(* Logix 5000 project; controller QW361 vendor 1 type 14 code 107 rev 32.11; software revision 32.00; part 11 of 20 *)

        [1429].time.Year := 2022, [1429].time.Month := 4, [1429].time.Day := 28, [1429].time.Hour := 20, [1429].time.Minute := 39, [1429].time.Second := 59, [1429].time.DST_ON := 1, [1430].log_data[0].min := 1.0, [1430].log_data[0].max := 1.0, [1430].log_data[0].total := 300.0, [1430].log_data[0].time := 300.0, [1430].log_data[0].minminute := 40, [1430].log_data[0].maxminute := 40, [1430].log_data[0].valid := 1, [1430].log_data[1].valid := 1, [1430].log_data[2].valid := 1, [1430].log_data[3].valid := 1, [1430].log_data[4].valid := 1, [1430].time.Year := 2022, [1430].time.Month := 4, [1430].time.Day := 28, [1430].time.Hour := 20, [1430].time.Minute := 44, [1430].time.Second := 59, [1430].time.DST_ON := 1, [1431].log_data[0].min := 1.0, [1431].log_data[0].max := 1.0, [1431].log_data[0].total := 300.0, [1431].log_data[0].time := 300.0, [1431].log_data[0].minminute := 45, [1431].log_data[0].maxminute := 45, [1431].log_data[0].valid := 1, [1431].log_data[1].valid := 1, [1431].log_data[2].valid := 1, [1431].log_data[3].valid := 1, [1431].log_data[4].valid := 1, [1431].time.Year := 2022, [1431].time.Month := 4, [1431].time.Day := 28, [1431].time.Hour := 20, [1431].time.Minute := 49, [1431].time.Second := 59, [1431].time.DST_ON := 1, [1432].log_data[0].min := 1.0, [1432].log_data[0].max := 1.0, [1432].log_data[0].total := 300.0, [1432].log_data[0].time := 300.0, [1432].log_data[0].minminute := 50, [1432].log_data[0].maxminute := 50, [1432].log_data[0].valid := 1, [1432].log_data[1].valid := 1, [1432].log_data[2].valid := 1, [1432].log_data[3].valid := 1, [1432].log_data[4].valid := 1, [1432].time.Year := 2022, [1432].time.Month := 4, [1432].time.Day := 28, [1432].time.Hour := 20, [1432].time.Minute := 54, [1432].time.Second := 59,
        [1432].time.DST_ON := 1, [1433].log_data[0].min := 1.0, [1433].log_data[0].max := 1.0, [1433].log_data[0].total := 300.0, [1433].log_data[0].time := 300.0, [1433].log_data[0].minminute := 55, [1433].log_data[0].maxminute := 55, [1433].log_data[0].valid := 1, [1433].log_data[1].valid := 1, [1433].log_data[2].valid := 1, [1433].log_data[3].valid := 1, [1433].log_data[4].valid := 1, [1433].time.Year := 2022, [1433].time.Month := 4, [1433].time.Day := 28, [1433].time.Hour := 20, [1433].time.Minute := 59, [1433].time.Second := 59, [1433].time.DST_ON := 1, [1434].log_data[0].min := 1.0, [1434].log_data[0].max := 1.0, [1434].log_data[0].total := 300.0, [1434].log_data[0].time := 300.0, [1434].log_data[0].valid := 1, [1434].log_data[1].valid := 1, [1434].log_data[2].valid := 1, [1434].log_data[3].valid := 1, [1434].log_data[4].valid := 1, [1434].time.Year := 2022, [1434].time.Month := 4, [1434].time.Day := 28, [1434].time.Hour := 21, [1434].time.Minute := 4, [1434].time.Second := 59, [1434].time.DST_ON := 1, [1435].log_data[0].min := 1.0, [1435].log_data[0].max := 1.0, [1435].log_data[0].total := 300.0, [1435].log_data[0].time := 300.0, [1435].log_data[0].minminute := 5, [1435].log_data[0].maxminute := 5, [1435].log_data[0].valid := 1, [1435].log_data[1].valid := 1, [1435].log_data[2].valid := 1, [1435].log_data[3].valid := 1, [1435].log_data[4].valid := 1, [1435].time.Year := 2022, [1435].time.Month := 4, [1435].time.Day := 28, [1435].time.Hour := 21, [1435].time.Minute := 9, [1435].time.Second := 59, [1435].time.DST_ON := 1, [1436].log_data[0].min := 1.0, [1436].log_data[0].max := 1.0, [1436].log_data[0].total := 300.0, [1436].log_data[0].time := 300.0, [1436].log_data[0].minminute := 10, [1436].log_data[0].maxminute := 10, [1436].log_data[0].valid := 1,
        [1436].log_data[1].valid := 1, [1436].log_data[2].valid := 1, [1436].log_data[3].valid := 1, [1436].log_data[4].valid := 1, [1436].time.Year := 2022, [1436].time.Month := 4, [1436].time.Day := 28, [1436].time.Hour := 21, [1436].time.Minute := 14, [1436].time.Second := 59, [1436].time.DST_ON := 1, [1437].log_data[0].min := 1.0, [1437].log_data[0].max := 1.0, [1437].log_data[0].total := 300.0, [1437].log_data[0].time := 300.0, [1437].log_data[0].minminute := 15, [1437].log_data[0].maxminute := 15, [1437].log_data[0].valid := 1, [1437].log_data[1].valid := 1, [1437].log_data[2].valid := 1, [1437].log_data[3].valid := 1, [1437].log_data[4].valid := 1, [1437].time.Year := 2022, [1437].time.Month := 4, [1437].time.Day := 28, [1437].time.Hour := 21, [1437].time.Minute := 19, [1437].time.Second := 59, [1437].time.DST_ON := 1, [1438].log_data[0].min := 1.0, [1438].log_data[0].max := 1.0, [1438].log_data[0].total := 300.0, [1438].log_data[0].time := 300.0, [1438].log_data[0].minminute := 20, [1438].log_data[0].maxminute := 20, [1438].log_data[0].valid := 1, [1438].log_data[1].valid := 1, [1438].log_data[2].valid := 1, [1438].log_data[3].valid := 1, [1438].log_data[4].valid := 1, [1438].time.Year := 2022, [1438].time.Month := 4, [1438].time.Day := 28, [1438].time.Hour := 21, [1438].time.Minute := 24, [1438].time.Second := 59, [1438].time.DST_ON := 1, [1439].log_data[0].min := 1.0, [1439].log_data[0].max := 1.0, [1439].log_data[0].total := 300.0, [1439].log_data[0].time := 300.0, [1439].log_data[0].minminute := 25, [1439].log_data[0].maxminute := 25, [1439].log_data[0].valid := 1, [1439].log_data[1].valid := 1, [1439].log_data[2].valid := 1, [1439].log_data[3].valid := 1, [1439].log_data[4].valid := 1, [1439].time.Year := 2022, [1439].time.Month := 4,
        [1439].time.Day := 28, [1439].time.Hour := 21, [1439].time.Minute := 29, [1439].time.Second := 59, [1439].time.DST_ON := 1, [1440].log_data[0].min := 1.0, [1440].log_data[0].max := 1.0, [1440].log_data[0].total := 300.0, [1440].log_data[0].time := 300.0, [1440].log_data[0].minminute := 30, [1440].log_data[0].maxminute := 30, [1440].log_data[0].valid := 1, [1440].log_data[1].valid := 1, [1440].log_data[2].valid := 1, [1440].log_data[3].valid := 1, [1440].log_data[4].valid := 1, [1440].time.Year := 2022, [1440].time.Month := 4, [1440].time.Day := 28, [1440].time.Hour := 21, [1440].time.Minute := 34, [1440].time.Second := 59, [1440].time.DST_ON := 1, [1441].log_data[0].min := 1.0, [1441].log_data[0].max := 1.0, [1441].log_data[0].total := 300.0, [1441].log_data[0].time := 300.0, [1441].log_data[0].minminute := 35, [1441].log_data[0].maxminute := 35, [1441].log_data[0].valid := 1, [1441].log_data[1].valid := 1, [1441].log_data[2].valid := 1, [1441].log_data[3].valid := 1, [1441].log_data[4].valid := 1, [1441].time.Year := 2022, [1441].time.Month := 4, [1441].time.Day := 28, [1441].time.Hour := 21, [1441].time.Minute := 39, [1441].time.Second := 59, [1441].time.DST_ON := 1, [1442].log_data[0].min := 1.0, [1442].log_data[0].max := 1.0, [1442].log_data[0].total := 300.0, [1442].log_data[0].time := 300.0, [1442].log_data[0].minminute := 40, [1442].log_data[0].maxminute := 40, [1442].log_data[0].valid := 1, [1442].log_data[1].valid := 1, [1442].log_data[2].valid := 1, [1442].log_data[3].valid := 1, [1442].log_data[4].valid := 1, [1442].time.Year := 2022, [1442].time.Month := 4, [1442].time.Day := 28, [1442].time.Hour := 21, [1442].time.Minute := 44, [1442].time.Second := 59, [1442].time.DST_ON := 1, [1443].log_data[0].min := 1.0,
        [1443].log_data[0].max := 1.0, [1443].log_data[0].total := 300.0, [1443].log_data[0].time := 300.0, [1443].log_data[0].minminute := 45, [1443].log_data[0].maxminute := 45, [1443].log_data[0].valid := 1, [1443].log_data[1].valid := 1, [1443].log_data[2].valid := 1, [1443].log_data[3].valid := 1, [1443].log_data[4].valid := 1, [1443].time.Year := 2022, [1443].time.Month := 4, [1443].time.Day := 28, [1443].time.Hour := 21, [1443].time.Minute := 49, [1443].time.Second := 59, [1443].time.DST_ON := 1, [1444].log_data[0].min := 1.0, [1444].log_data[0].max := 1.0, [1444].log_data[0].total := 300.0, [1444].log_data[0].time := 300.0, [1444].log_data[0].minminute := 50, [1444].log_data[0].maxminute := 50, [1444].log_data[0].valid := 1, [1444].log_data[1].valid := 1, [1444].log_data[2].valid := 1, [1444].log_data[3].valid := 1, [1444].log_data[4].valid := 1, [1444].time.Year := 2022, [1444].time.Month := 4, [1444].time.Day := 28, [1444].time.Hour := 21, [1444].time.Minute := 54, [1444].time.Second := 59, [1444].time.DST_ON := 1, [1445].log_data[0].min := 1.0, [1445].log_data[0].max := 1.0, [1445].log_data[0].total := 300.0, [1445].log_data[0].time := 300.0, [1445].log_data[0].minminute := 55, [1445].log_data[0].maxminute := 55, [1445].log_data[0].valid := 1, [1445].log_data[1].valid := 1, [1445].log_data[2].valid := 1, [1445].log_data[3].valid := 1, [1445].log_data[4].valid := 1, [1445].time.Year := 2022, [1445].time.Month := 4, [1445].time.Day := 28, [1445].time.Hour := 21, [1445].time.Minute := 59, [1445].time.Second := 59, [1445].time.DST_ON := 1, [1446].log_data[0].min := 1.0, [1446].log_data[0].max := 1.0, [1446].log_data[0].total := 300.0, [1446].log_data[0].time := 300.0, [1446].log_data[0].valid := 1, [1446].log_data[1].valid := 1, [1446].log_data[2].valid := 1,
        [1446].log_data[3].valid := 1, [1446].log_data[4].valid := 1, [1446].time.Year := 2022, [1446].time.Month := 4, [1446].time.Day := 28, [1446].time.Hour := 22, [1446].time.Minute := 4, [1446].time.Second := 59, [1446].time.DST_ON := 1, [1447].log_data[0].min := 1.0, [1447].log_data[0].max := 1.0, [1447].log_data[0].total := 300.0, [1447].log_data[0].time := 300.0, [1447].log_data[0].minminute := 5, [1447].log_data[0].maxminute := 5, [1447].log_data[0].valid := 1, [1447].log_data[1].valid := 1, [1447].log_data[2].valid := 1, [1447].log_data[3].valid := 1, [1447].log_data[4].valid := 1, [1447].time.Year := 2022, [1447].time.Month := 4, [1447].time.Day := 28, [1447].time.Hour := 22, [1447].time.Minute := 9, [1447].time.Second := 59, [1447].time.DST_ON := 1, [1448].log_data[0].min := 1.0, [1448].log_data[0].max := 1.0, [1448].log_data[0].total := 300.0, [1448].log_data[0].time := 300.0, [1448].log_data[0].minminute := 10, [1448].log_data[0].maxminute := 10, [1448].log_data[0].valid := 1, [1448].log_data[1].valid := 1, [1448].log_data[2].valid := 1, [1448].log_data[3].valid := 1, [1448].log_data[4].valid := 1, [1448].time.Year := 2022, [1448].time.Month := 4, [1448].time.Day := 28, [1448].time.Hour := 22, [1448].time.Minute := 14, [1448].time.Second := 59, [1448].time.DST_ON := 1, [1449].log_data[0].min := 1.0, [1449].log_data[0].max := 1.0, [1449].log_data[0].total := 300.0, [1449].log_data[0].time := 300.0, [1449].log_data[0].minminute := 15, [1449].log_data[0].maxminute := 15, [1449].log_data[0].valid := 1, [1449].log_data[1].valid := 1, [1449].log_data[2].valid := 1, [1449].log_data[3].valid := 1, [1449].log_data[4].valid := 1, [1449].time.Year := 2022, [1449].time.Month := 4, [1449].time.Day := 28, [1449].time.Hour := 22,
        [1449].time.Minute := 19, [1449].time.Second := 59, [1449].time.DST_ON := 1, [1450].log_data[0].min := 1.0, [1450].log_data[0].max := 1.0, [1450].log_data[0].total := 300.0, [1450].log_data[0].time := 300.0, [1450].log_data[0].minminute := 20, [1450].log_data[0].maxminute := 20, [1450].log_data[0].valid := 1, [1450].log_data[1].valid := 1, [1450].log_data[2].valid := 1, [1450].log_data[3].valid := 1, [1450].log_data[4].valid := 1, [1450].time.Year := 2022, [1450].time.Month := 4, [1450].time.Day := 28, [1450].time.Hour := 22, [1450].time.Minute := 24, [1450].time.Second := 59, [1450].time.DST_ON := 1, [1451].log_data[0].min := 1.0, [1451].log_data[0].max := 1.0, [1451].log_data[0].total := 300.0, [1451].log_data[0].time := 300.0, [1451].log_data[0].minminute := 25, [1451].log_data[0].maxminute := 25, [1451].log_data[0].valid := 1, [1451].log_data[1].valid := 1, [1451].log_data[2].valid := 1, [1451].log_data[3].valid := 1, [1451].log_data[4].valid := 1, [1451].time.Year := 2022, [1451].time.Month := 4, [1451].time.Day := 28, [1451].time.Hour := 22, [1451].time.Minute := 29, [1451].time.Second := 59, [1451].time.DST_ON := 1, [1452].log_data[0].min := 1.0, [1452].log_data[0].max := 1.0, [1452].log_data[0].total := 300.0, [1452].log_data[0].time := 300.0, [1452].log_data[0].minminute := 30, [1452].log_data[0].maxminute := 30, [1452].log_data[0].valid := 1, [1452].log_data[1].valid := 1, [1452].log_data[2].valid := 1, [1452].log_data[3].valid := 1, [1452].log_data[4].valid := 1, [1452].time.Year := 2022, [1452].time.Month := 4, [1452].time.Day := 28, [1452].time.Hour := 22, [1452].time.Minute := 34, [1452].time.Second := 59, [1452].time.DST_ON := 1, [1453].log_data[0].min := 1.0, [1453].log_data[0].max := 1.0, [1453].log_data[0].total := 300.0,
        [1453].log_data[0].time := 300.0, [1453].log_data[0].minminute := 35, [1453].log_data[0].maxminute := 35, [1453].log_data[0].valid := 1, [1453].log_data[1].valid := 1, [1453].log_data[2].valid := 1, [1453].log_data[3].valid := 1, [1453].log_data[4].valid := 1, [1453].time.Year := 2022, [1453].time.Month := 4, [1453].time.Day := 28, [1453].time.Hour := 22, [1453].time.Minute := 39, [1453].time.Second := 59, [1453].time.DST_ON := 1, [1454].log_data[0].min := 1.0, [1454].log_data[0].max := 1.0, [1454].log_data[0].total := 300.0, [1454].log_data[0].time := 300.0, [1454].log_data[0].minminute := 40, [1454].log_data[0].maxminute := 40, [1454].log_data[0].valid := 1, [1454].log_data[1].valid := 1, [1454].log_data[2].valid := 1, [1454].log_data[3].valid := 1, [1454].log_data[4].valid := 1, [1454].time.Year := 2022, [1454].time.Month := 4, [1454].time.Day := 28, [1454].time.Hour := 22, [1454].time.Minute := 44, [1454].time.Second := 59, [1454].time.DST_ON := 1, [1455].log_data[0].min := 1.0, [1455].log_data[0].max := 1.0, [1455].log_data[0].total := 300.0, [1455].log_data[0].time := 300.0, [1455].log_data[0].minminute := 45, [1455].log_data[0].maxminute := 45, [1455].log_data[0].valid := 1, [1455].log_data[1].valid := 1, [1455].log_data[2].valid := 1, [1455].log_data[3].valid := 1, [1455].log_data[4].valid := 1, [1455].time.Year := 2022, [1455].time.Month := 4, [1455].time.Day := 28, [1455].time.Hour := 22, [1455].time.Minute := 49, [1455].time.Second := 59, [1455].time.DST_ON := 1, [1456].log_data[0].min := 1.0, [1456].log_data[0].max := 1.0, [1456].log_data[0].total := 300.0, [1456].log_data[0].time := 300.0, [1456].log_data[0].minminute := 50, [1456].log_data[0].maxminute := 50, [1456].log_data[0].valid := 1, [1456].log_data[1].valid := 1, [1456].log_data[2].valid := 1,
        [1456].log_data[3].valid := 1, [1456].log_data[4].valid := 1, [1456].time.Year := 2022, [1456].time.Month := 4, [1456].time.Day := 28, [1456].time.Hour := 22, [1456].time.Minute := 54, [1456].time.Second := 59, [1456].time.DST_ON := 1, [1457].log_data[0].min := 1.0, [1457].log_data[0].max := 1.0, [1457].log_data[0].total := 300.0, [1457].log_data[0].time := 300.0, [1457].log_data[0].minminute := 55, [1457].log_data[0].maxminute := 55, [1457].log_data[0].valid := 1, [1457].log_data[1].valid := 1, [1457].log_data[2].valid := 1, [1457].log_data[3].valid := 1, [1457].log_data[4].valid := 1, [1457].time.Year := 2022, [1457].time.Month := 4, [1457].time.Day := 28, [1457].time.Hour := 22, [1457].time.Minute := 59, [1457].time.Second := 59, [1457].time.DST_ON := 1, [1458].log_data[0].min := 1.0, [1458].log_data[0].max := 1.0, [1458].log_data[0].total := 300.0, [1458].log_data[0].time := 300.0, [1458].log_data[0].valid := 1, [1458].log_data[1].valid := 1, [1458].log_data[2].valid := 1, [1458].log_data[3].valid := 1, [1458].log_data[4].valid := 1, [1458].time.Year := 2022, [1458].time.Month := 4, [1458].time.Day := 28, [1458].time.Hour := 23, [1458].time.Minute := 4, [1458].time.Second := 59, [1458].time.DST_ON := 1, [1459].log_data[0].min := 1.0, [1459].log_data[0].max := 1.0, [1459].log_data[0].total := 300.0, [1459].log_data[0].time := 300.0, [1459].log_data[0].minminute := 5, [1459].log_data[0].maxminute := 5, [1459].log_data[0].valid := 1, [1459].log_data[1].valid := 1, [1459].log_data[2].valid := 1, [1459].log_data[3].valid := 1, [1459].log_data[4].valid := 1, [1459].time.Year := 2022, [1459].time.Month := 4, [1459].time.Day := 28, [1459].time.Hour := 23, [1459].time.Minute := 9, [1459].time.Second := 59,
        [1459].time.DST_ON := 1, [1460].log_data[0].min := 1.0, [1460].log_data[0].max := 1.0, [1460].log_data[0].total := 300.0, [1460].log_data[0].time := 300.0, [1460].log_data[0].minminute := 10, [1460].log_data[0].maxminute := 10, [1460].log_data[0].valid := 1, [1460].log_data[1].valid := 1, [1460].log_data[2].valid := 1, [1460].log_data[3].valid := 1, [1460].log_data[4].valid := 1, [1460].time.Year := 2022, [1460].time.Month := 4, [1460].time.Day := 28, [1460].time.Hour := 23, [1460].time.Minute := 14, [1460].time.Second := 59, [1460].time.DST_ON := 1, [1461].log_data[0].min := 1.0, [1461].log_data[0].max := 1.0, [1461].log_data[0].total := 300.0, [1461].log_data[0].time := 300.0, [1461].log_data[0].minminute := 15, [1461].log_data[0].maxminute := 15, [1461].log_data[0].valid := 1, [1461].log_data[1].valid := 1, [1461].log_data[2].valid := 1, [1461].log_data[3].valid := 1, [1461].log_data[4].valid := 1, [1461].time.Year := 2022, [1461].time.Month := 4, [1461].time.Day := 28, [1461].time.Hour := 23, [1461].time.Minute := 19, [1461].time.Second := 59, [1461].time.DST_ON := 1, [1462].log_data[0].min := 1.0, [1462].log_data[0].max := 1.0, [1462].log_data[0].total := 300.0, [1462].log_data[0].time := 300.0, [1462].log_data[0].minminute := 20, [1462].log_data[0].maxminute := 20, [1462].log_data[0].valid := 1, [1462].log_data[1].valid := 1, [1462].log_data[2].valid := 1, [1462].log_data[3].valid := 1, [1462].log_data[4].valid := 1, [1462].time.Year := 2022, [1462].time.Month := 4, [1462].time.Day := 28, [1462].time.Hour := 23, [1462].time.Minute := 24, [1462].time.Second := 59, [1462].time.DST_ON := 1, [1463].log_data[0].min := 1.0, [1463].log_data[0].max := 1.0, [1463].log_data[0].total := 300.0, [1463].log_data[0].time := 300.0, [1463].log_data[0].minminute := 25,
        [1463].log_data[0].maxminute := 25, [1463].log_data[0].valid := 1, [1463].log_data[1].valid := 1, [1463].log_data[2].valid := 1, [1463].log_data[3].valid := 1, [1463].log_data[4].valid := 1, [1463].time.Year := 2022, [1463].time.Month := 4, [1463].time.Day := 28, [1463].time.Hour := 23, [1463].time.Minute := 29, [1463].time.Second := 59, [1463].time.DST_ON := 1, [1464].log_data[0].min := 1.0, [1464].log_data[0].max := 1.0, [1464].log_data[0].total := 300.0, [1464].log_data[0].time := 300.0, [1464].log_data[0].minminute := 30, [1464].log_data[0].maxminute := 30, [1464].log_data[0].valid := 1, [1464].log_data[1].valid := 1, [1464].log_data[2].valid := 1, [1464].log_data[3].valid := 1, [1464].log_data[4].valid := 1, [1464].time.Year := 2022, [1464].time.Month := 4, [1464].time.Day := 28, [1464].time.Hour := 23, [1464].time.Minute := 34, [1464].time.Second := 59, [1464].time.DST_ON := 1, [1465].log_data[0].min := 1.0, [1465].log_data[0].max := 1.0, [1465].log_data[0].total := 300.0, [1465].log_data[0].time := 300.0, [1465].log_data[0].minminute := 35, [1465].log_data[0].maxminute := 35, [1465].log_data[0].valid := 1, [1465].log_data[1].valid := 1, [1465].log_data[2].valid := 1, [1465].log_data[3].valid := 1, [1465].log_data[4].valid := 1, [1465].time.Year := 2022, [1465].time.Month := 4, [1465].time.Day := 28, [1465].time.Hour := 23, [1465].time.Minute := 39, [1465].time.Second := 59, [1465].time.DST_ON := 1, [1466].log_data[0].min := 1.0, [1466].log_data[0].max := 1.0, [1466].log_data[0].total := 300.0, [1466].log_data[0].time := 300.0, [1466].log_data[0].minminute := 40, [1466].log_data[0].maxminute := 40, [1466].log_data[0].valid := 1, [1466].log_data[1].valid := 1, [1466].log_data[2].valid := 1, [1466].log_data[3].valid := 1, [1466].log_data[4].valid := 1,
        [1466].time.Year := 2022, [1466].time.Month := 4, [1466].time.Day := 28, [1466].time.Hour := 23, [1466].time.Minute := 44, [1466].time.Second := 59, [1466].time.DST_ON := 1, [1467].log_data[0].min := 1.0, [1467].log_data[0].max := 1.0, [1467].log_data[0].total := 300.0, [1467].log_data[0].time := 300.0, [1467].log_data[0].minminute := 45, [1467].log_data[0].maxminute := 45, [1467].log_data[0].valid := 1, [1467].log_data[1].valid := 1, [1467].log_data[2].valid := 1, [1467].log_data[3].valid := 1, [1467].log_data[4].valid := 1, [1467].time.Year := 2022, [1467].time.Month := 4, [1467].time.Day := 28, [1467].time.Hour := 23, [1467].time.Minute := 49, [1467].time.Second := 59, [1467].time.DST_ON := 1, [1468].log_data[0].min := 1.0, [1468].log_data[0].max := 1.0, [1468].log_data[0].total := 300.0, [1468].log_data[0].time := 300.0, [1468].log_data[0].minminute := 50, [1468].log_data[0].maxminute := 50, [1468].log_data[0].valid := 1, [1468].log_data[1].valid := 1, [1468].log_data[2].valid := 1, [1468].log_data[3].valid := 1, [1468].log_data[4].valid := 1, [1468].time.Year := 2022, [1468].time.Month := 4, [1468].time.Day := 28, [1468].time.Hour := 23, [1468].time.Minute := 54, [1468].time.Second := 59, [1468].time.DST_ON := 1, [1469].log_data[0].min := 1.0, [1469].log_data[0].max := 1.0, [1469].log_data[0].total := 300.0, [1469].log_data[0].time := 300.0, [1469].log_data[0].minminute := 55, [1469].log_data[0].maxminute := 55, [1469].log_data[0].valid := 1, [1469].log_data[1].valid := 1, [1469].log_data[2].valid := 1, [1469].log_data[3].valid := 1, [1469].log_data[4].valid := 1, [1469].time.Year := 2022, [1469].time.Month := 4, [1469].time.Day := 28, [1469].time.Hour := 23, [1469].time.Minute := 59, [1469].time.Second := 59,
        [1469].time.DST_ON := 1, [1470].log_data[0].min := 1.0, [1470].log_data[0].max := 1.0, [1470].log_data[0].total := 300.0, [1470].log_data[0].time := 300.0, [1470].log_data[0].valid := 1, [1470].log_data[1].valid := 1, [1470].log_data[2].valid := 1, [1470].log_data[3].valid := 1, [1470].log_data[4].valid := 1, [1470].time.Year := 2022, [1470].time.Month := 4, [1470].time.Day := 29, [1470].time.Minute := 4, [1470].time.Second := 59, [1470].time.DST_ON := 1, [1471].log_data[0].min := 1.0, [1471].log_data[0].max := 1.0, [1471].log_data[0].total := 300.0, [1471].log_data[0].time := 300.0, [1471].log_data[0].minminute := 5, [1471].log_data[0].maxminute := 5, [1471].log_data[0].valid := 1, [1471].log_data[1].valid := 1, [1471].log_data[2].valid := 1, [1471].log_data[3].valid := 1, [1471].log_data[4].valid := 1, [1471].time.Year := 2022, [1471].time.Month := 4, [1471].time.Day := 29, [1471].time.Minute := 9, [1471].time.Second := 59, [1471].time.DST_ON := 1, [1472].log_data[0].min := 1.0, [1472].log_data[0].max := 1.0, [1472].log_data[0].total := 300.0, [1472].log_data[0].time := 300.0, [1472].log_data[0].minminute := 10, [1472].log_data[0].maxminute := 10, [1472].log_data[0].valid := 1, [1472].log_data[1].valid := 1, [1472].log_data[2].valid := 1, [1472].log_data[3].valid := 1, [1472].log_data[4].valid := 1, [1472].time.Year := 2022, [1472].time.Month := 4, [1472].time.Day := 29, [1472].time.Minute := 14, [1472].time.Second := 59, [1472].time.DST_ON := 1, [1473].log_data[0].min := 1.0, [1473].log_data[0].max := 1.0, [1473].log_data[0].total := 300.0, [1473].log_data[0].time := 300.0, [1473].log_data[0].minminute := 15, [1473].log_data[0].maxminute := 15, [1473].log_data[0].valid := 1, [1473].log_data[1].valid := 1, [1473].log_data[2].valid := 1, [1473].log_data[3].valid := 1,
        [1473].log_data[4].valid := 1, [1473].time.Year := 2022, [1473].time.Month := 4, [1473].time.Day := 29, [1473].time.Minute := 19, [1473].time.Second := 59, [1473].time.DST_ON := 1, [1474].log_data[0].min := 1.0, [1474].log_data[0].max := 1.0, [1474].log_data[0].total := 300.0, [1474].log_data[0].time := 300.0, [1474].log_data[0].minminute := 20, [1474].log_data[0].maxminute := 20, [1474].log_data[0].valid := 1, [1474].log_data[1].valid := 1, [1474].log_data[2].valid := 1, [1474].log_data[3].valid := 1, [1474].log_data[4].valid := 1, [1474].time.Year := 2022, [1474].time.Month := 4, [1474].time.Day := 29, [1474].time.Minute := 24, [1474].time.Second := 59, [1474].time.DST_ON := 1, [1475].log_data[0].min := 1.0, [1475].log_data[0].max := 1.0, [1475].log_data[0].total := 300.0, [1475].log_data[0].time := 300.0, [1475].log_data[0].minminute := 25, [1475].log_data[0].maxminute := 25, [1475].log_data[0].valid := 1, [1475].log_data[1].valid := 1, [1475].log_data[2].valid := 1, [1475].log_data[3].valid := 1, [1475].log_data[4].valid := 1, [1475].time.Year := 2022, [1475].time.Month := 4, [1475].time.Day := 29, [1475].time.Minute := 29, [1475].time.Second := 59, [1475].time.DST_ON := 1, [1476].log_data[0].min := 1.0, [1476].log_data[0].max := 1.0, [1476].log_data[0].total := 300.0, [1476].log_data[0].time := 300.0, [1476].log_data[0].minminute := 30, [1476].log_data[0].maxminute := 30, [1476].log_data[0].valid := 1, [1476].log_data[1].valid := 1, [1476].log_data[2].valid := 1, [1476].log_data[3].valid := 1, [1476].log_data[4].valid := 1, [1476].time.Year := 2022, [1476].time.Month := 4, [1476].time.Day := 29, [1476].time.Minute := 34, [1476].time.Second := 59, [1476].time.DST_ON := 1, [1477].log_data[0].min := 1.0, [1477].log_data[0].max := 1.0,
        [1477].log_data[0].total := 300.0, [1477].log_data[0].time := 300.0, [1477].log_data[0].minminute := 35, [1477].log_data[0].maxminute := 35, [1477].log_data[0].valid := 1, [1477].log_data[1].valid := 1, [1477].log_data[2].valid := 1, [1477].log_data[3].valid := 1, [1477].log_data[4].valid := 1, [1477].time.Year := 2022, [1477].time.Month := 4, [1477].time.Day := 29, [1477].time.Minute := 39, [1477].time.Second := 59, [1477].time.DST_ON := 1, [1478].log_data[0].min := 1.0, [1478].log_data[0].max := 1.0, [1478].log_data[0].total := 300.0, [1478].log_data[0].time := 300.0, [1478].log_data[0].minminute := 40, [1478].log_data[0].maxminute := 40, [1478].log_data[0].valid := 1, [1478].log_data[1].valid := 1, [1478].log_data[2].valid := 1, [1478].log_data[3].valid := 1, [1478].log_data[4].valid := 1, [1478].time.Year := 2022, [1478].time.Month := 4, [1478].time.Day := 29, [1478].time.Minute := 44, [1478].time.Second := 59, [1478].time.DST_ON := 1, [1479].log_data[0].min := 1.0, [1479].log_data[0].max := 1.0, [1479].log_data[0].total := 300.0, [1479].log_data[0].time := 300.0, [1479].log_data[0].minminute := 45, [1479].log_data[0].maxminute := 45, [1479].log_data[0].valid := 1, [1479].log_data[1].valid := 1, [1479].log_data[2].valid := 1, [1479].log_data[3].valid := 1, [1479].log_data[4].valid := 1, [1479].time.Year := 2022, [1479].time.Month := 4, [1479].time.Day := 29, [1479].time.Minute := 49, [1479].time.Second := 59, [1479].time.DST_ON := 1, [1480].log_data[0].min := 1.0, [1480].log_data[0].max := 1.0, [1480].log_data[0].total := 300.0, [1480].log_data[0].time := 300.0, [1480].log_data[0].minminute := 50, [1480].log_data[0].maxminute := 50, [1480].log_data[0].valid := 1, [1480].log_data[1].valid := 1, [1480].log_data[2].valid := 1, [1480].log_data[3].valid := 1, [1480].log_data[4].valid := 1,
        [1480].time.Year := 2022, [1480].time.Month := 4, [1480].time.Day := 29, [1480].time.Minute := 54, [1480].time.Second := 59, [1480].time.DST_ON := 1, [1481].log_data[0].min := 1.0, [1481].log_data[0].max := 1.0, [1481].log_data[0].total := 300.0, [1481].log_data[0].time := 300.0, [1481].log_data[0].minminute := 55, [1481].log_data[0].maxminute := 55, [1481].log_data[0].valid := 1, [1481].log_data[1].valid := 1, [1481].log_data[2].valid := 1, [1481].log_data[3].valid := 1, [1481].log_data[4].valid := 1, [1481].time.Year := 2022, [1481].time.Month := 4, [1481].time.Day := 29, [1481].time.Minute := 59, [1481].time.Second := 59, [1481].time.DST_ON := 1, [1482].log_data[0].min := 1.0, [1482].log_data[0].max := 1.0, [1482].log_data[0].total := 300.0, [1482].log_data[0].time := 300.0, [1482].log_data[0].valid := 1, [1482].log_data[1].valid := 1, [1482].log_data[2].valid := 1, [1482].log_data[3].valid := 1, [1482].log_data[4].valid := 1, [1482].time.Year := 2022, [1482].time.Month := 4, [1482].time.Day := 29, [1482].time.Hour := 1, [1482].time.Minute := 4, [1482].time.Second := 59, [1482].time.DST_ON := 1, [1483].log_data[0].min := 1.0, [1483].log_data[0].max := 1.0, [1483].log_data[0].total := 300.0, [1483].log_data[0].time := 300.0, [1483].log_data[0].minminute := 5, [1483].log_data[0].maxminute := 5, [1483].log_data[0].valid := 1, [1483].log_data[1].valid := 1, [1483].log_data[2].valid := 1, [1483].log_data[3].valid := 1, [1483].log_data[4].valid := 1, [1483].time.Year := 2022, [1483].time.Month := 4, [1483].time.Day := 29, [1483].time.Hour := 1, [1483].time.Minute := 9, [1483].time.Second := 59, [1483].time.DST_ON := 1, [1484].log_data[0].min := 1.0, [1484].log_data[0].max := 1.0, [1484].log_data[0].total := 300.0,
        [1484].log_data[0].time := 300.0, [1484].log_data[0].minminute := 10, [1484].log_data[0].maxminute := 10, [1484].log_data[0].valid := 1, [1484].log_data[1].valid := 1, [1484].log_data[2].valid := 1, [1484].log_data[3].valid := 1, [1484].log_data[4].valid := 1, [1484].time.Year := 2022, [1484].time.Month := 4, [1484].time.Day := 29, [1484].time.Hour := 1, [1484].time.Minute := 14, [1484].time.Second := 59, [1484].time.DST_ON := 1, [1485].log_data[0].min := 1.0, [1485].log_data[0].max := 1.0, [1485].log_data[0].total := 299.999, [1485].log_data[0].time := 299.999, [1485].log_data[0].minminute := 15, [1485].log_data[0].maxminute := 15, [1485].log_data[0].valid := 1, [1485].log_data[1].valid := 1, [1485].log_data[2].valid := 1, [1485].log_data[3].valid := 1, [1485].log_data[4].valid := 1, [1485].time.Year := 2022, [1485].time.Month := 4, [1485].time.Day := 29, [1485].time.Hour := 1, [1485].time.Minute := 19, [1485].time.Second := 59, [1485].time.DST_ON := 1, [1486].log_data[0].min := 1.0, [1486].log_data[0].max := 1.0, [1486].log_data[0].total := 300.0, [1486].log_data[0].time := 300.0, [1486].log_data[0].minminute := 20, [1486].log_data[0].maxminute := 20, [1486].log_data[0].valid := 1, [1486].log_data[1].valid := 1, [1486].log_data[2].valid := 1, [1486].log_data[3].valid := 1, [1486].log_data[4].valid := 1, [1486].time.Year := 2022, [1486].time.Month := 4, [1486].time.Day := 29, [1486].time.Hour := 1, [1486].time.Minute := 24, [1486].time.Second := 59, [1486].time.DST_ON := 1, [1487].log_data[0].min := 1.0, [1487].log_data[0].max := 1.0, [1487].log_data[0].total := 300.0, [1487].log_data[0].time := 300.0, [1487].log_data[0].minminute := 25, [1487].log_data[0].maxminute := 25, [1487].log_data[0].valid := 1, [1487].log_data[1].valid := 1, [1487].log_data[2].valid := 1,
        [1487].log_data[3].valid := 1, [1487].log_data[4].valid := 1, [1487].time.Year := 2022, [1487].time.Month := 4, [1487].time.Day := 29, [1487].time.Hour := 1, [1487].time.Minute := 29, [1487].time.Second := 59, [1487].time.DST_ON := 1, [1488].log_data[0].min := 1.0, [1488].log_data[0].max := 1.0, [1488].log_data[0].total := 300.0, [1488].log_data[0].time := 300.0, [1488].log_data[0].minminute := 30, [1488].log_data[0].maxminute := 30, [1488].log_data[0].valid := 1, [1488].log_data[1].valid := 1, [1488].log_data[2].valid := 1, [1488].log_data[3].valid := 1, [1488].log_data[4].valid := 1, [1488].time.Year := 2022, [1488].time.Month := 4, [1488].time.Day := 29, [1488].time.Hour := 1, [1488].time.Minute := 34, [1488].time.Second := 59, [1488].time.DST_ON := 1, [1489].log_data[0].min := 1.0, [1489].log_data[0].max := 1.0, [1489].log_data[0].total := 300.0, [1489].log_data[0].time := 300.0, [1489].log_data[0].minminute := 35, [1489].log_data[0].maxminute := 35, [1489].log_data[0].valid := 1, [1489].log_data[1].valid := 1, [1489].log_data[2].valid := 1, [1489].log_data[3].valid := 1, [1489].log_data[4].valid := 1, [1489].time.Year := 2022, [1489].time.Month := 4, [1489].time.Day := 29, [1489].time.Hour := 1, [1489].time.Minute := 39, [1489].time.Second := 59, [1489].time.DST_ON := 1, [1490].log_data[0].min := 1.0, [1490].log_data[0].max := 1.0, [1490].log_data[0].total := 299.999, [1490].log_data[0].time := 299.999, [1490].log_data[0].minminute := 40, [1490].log_data[0].maxminute := 40, [1490].log_data[0].valid := 1, [1490].log_data[1].valid := 1, [1490].log_data[2].valid := 1, [1490].log_data[3].valid := 1, [1490].log_data[4].valid := 1, [1490].time.Year := 2022, [1490].time.Month := 4, [1490].time.Day := 29, [1490].time.Hour := 1,
        [1490].time.Minute := 44, [1490].time.Second := 59, [1490].time.DST_ON := 1, [1491].log_data[0].min := 1.0, [1491].log_data[0].max := 1.0, [1491].log_data[0].total := 300.0, [1491].log_data[0].time := 300.0, [1491].log_data[0].minminute := 45, [1491].log_data[0].maxminute := 45, [1491].log_data[0].valid := 1, [1491].log_data[1].valid := 1, [1491].log_data[2].valid := 1, [1491].log_data[3].valid := 1, [1491].log_data[4].valid := 1, [1491].time.Year := 2022, [1491].time.Month := 4, [1491].time.Day := 29, [1491].time.Hour := 1, [1491].time.Minute := 49, [1491].time.Second := 59, [1491].time.DST_ON := 1, [1492].log_data[0].min := 1.0, [1492].log_data[0].max := 1.0, [1492].log_data[0].total := 300.0, [1492].log_data[0].time := 300.0, [1492].log_data[0].minminute := 50, [1492].log_data[0].maxminute := 50, [1492].log_data[0].valid := 1, [1492].log_data[1].valid := 1, [1492].log_data[2].valid := 1, [1492].log_data[3].valid := 1, [1492].log_data[4].valid := 1, [1492].time.Year := 2022, [1492].time.Month := 4, [1492].time.Day := 29, [1492].time.Hour := 1, [1492].time.Minute := 54, [1492].time.Second := 59, [1492].time.DST_ON := 1, [1493].log_data[0].min := 1.0, [1493].log_data[0].max := 1.0, [1493].log_data[0].total := 300.0, [1493].log_data[0].time := 300.0, [1493].log_data[0].minminute := 55, [1493].log_data[0].maxminute := 55, [1493].log_data[0].valid := 1, [1493].log_data[1].valid := 1, [1493].log_data[2].valid := 1, [1493].log_data[3].valid := 1, [1493].log_data[4].valid := 1, [1493].time.Year := 2022, [1493].time.Month := 4, [1493].time.Day := 29, [1493].time.Hour := 1, [1493].time.Minute := 59, [1493].time.Second := 59, [1493].time.DST_ON := 1, [1494].log_data[0].min := 1.0, [1494].log_data[0].max := 1.0, [1494].log_data[0].total := 300.0,
        [1494].log_data[0].time := 300.0, [1494].log_data[0].valid := 1, [1494].log_data[1].valid := 1, [1494].log_data[2].valid := 1, [1494].log_data[3].valid := 1, [1494].log_data[4].valid := 1, [1494].time.Year := 2022, [1494].time.Month := 4, [1494].time.Day := 29, [1494].time.Hour := 2, [1494].time.Minute := 4, [1494].time.Second := 59, [1494].time.DST_ON := 1, [1495].log_data[0].min := 1.0, [1495].log_data[0].max := 1.0, [1495].log_data[0].total := 300.0, [1495].log_data[0].time := 300.0, [1495].log_data[0].minminute := 5, [1495].log_data[0].maxminute := 5, [1495].log_data[0].valid := 1, [1495].log_data[1].valid := 1, [1495].log_data[2].valid := 1, [1495].log_data[3].valid := 1, [1495].log_data[4].valid := 1, [1495].time.Year := 2022, [1495].time.Month := 4, [1495].time.Day := 29, [1495].time.Hour := 2, [1495].time.Minute := 9, [1495].time.Second := 59, [1495].time.DST_ON := 1, [1496].log_data[0].min := 1.0, [1496].log_data[0].max := 1.0, [1496].log_data[0].total := 300.0, [1496].log_data[0].time := 300.0, [1496].log_data[0].minminute := 10, [1496].log_data[0].maxminute := 10, [1496].log_data[0].valid := 1, [1496].log_data[1].valid := 1, [1496].log_data[2].valid := 1, [1496].log_data[3].valid := 1, [1496].log_data[4].valid := 1, [1496].time.Year := 2022, [1496].time.Month := 4, [1496].time.Day := 29, [1496].time.Hour := 2, [1496].time.Minute := 14, [1496].time.Second := 59, [1496].time.DST_ON := 1, [1497].log_data[0].min := 1.0, [1497].log_data[0].max := 1.0, [1497].log_data[0].total := 300.0, [1497].log_data[0].time := 300.0, [1497].log_data[0].minminute := 15, [1497].log_data[0].maxminute := 15, [1497].log_data[0].valid := 1, [1497].log_data[1].valid := 1, [1497].log_data[2].valid := 1, [1497].log_data[3].valid := 1, [1497].log_data[4].valid := 1,
        [1497].time.Year := 2022, [1497].time.Month := 4, [1497].time.Day := 29, [1497].time.Hour := 2, [1497].time.Minute := 19, [1497].time.Second := 59, [1497].time.DST_ON := 1, [1498].log_data[0].min := 1.0, [1498].log_data[0].max := 1.0, [1498].log_data[0].total := 300.0, [1498].log_data[0].time := 300.0, [1498].log_data[0].minminute := 20, [1498].log_data[0].maxminute := 20, [1498].log_data[0].valid := 1, [1498].log_data[1].valid := 1, [1498].log_data[2].valid := 1, [1498].log_data[3].valid := 1, [1498].log_data[4].valid := 1, [1498].time.Year := 2022, [1498].time.Month := 4, [1498].time.Day := 29, [1498].time.Hour := 2, [1498].time.Minute := 24, [1498].time.Second := 59, [1498].time.DST_ON := 1, [1499].log_data[0].min := 1.0, [1499].log_data[0].max := 1.0, [1499].log_data[0].total := 300.0, [1499].log_data[0].time := 300.0, [1499].log_data[0].minminute := 25, [1499].log_data[0].maxminute := 25, [1499].log_data[0].valid := 1, [1499].log_data[1].valid := 1, [1499].log_data[2].valid := 1, [1499].log_data[3].valid := 1, [1499].log_data[4].valid := 1, [1499].time.Year := 2022, [1499].time.Month := 4, [1499].time.Day := 29, [1499].time.Hour := 2, [1499].time.Minute := 29, [1499].time.Second := 59, [1499].time.DST_ON := 1, [1500].log_data[0].min := 1.0, [1500].log_data[0].max := 1.0, [1500].log_data[0].total := 300.0, [1500].log_data[0].time := 300.0, [1500].log_data[0].minminute := 30, [1500].log_data[0].maxminute := 30, [1500].log_data[0].valid := 1, [1500].log_data[1].valid := 1, [1500].log_data[2].valid := 1, [1500].log_data[3].valid := 1, [1500].log_data[4].valid := 1, [1500].time.Year := 2022, [1500].time.Month := 4, [1500].time.Day := 29, [1500].time.Hour := 2, [1500].time.Minute := 34, [1500].time.Second := 59,
        [1500].time.DST_ON := 1, [1501].log_data[0].min := 1.0, [1501].log_data[0].max := 1.0, [1501].log_data[0].total := 300.0, [1501].log_data[0].time := 300.0, [1501].log_data[0].minminute := 35, [1501].log_data[0].maxminute := 35, [1501].log_data[0].valid := 1, [1501].log_data[1].valid := 1, [1501].log_data[2].valid := 1, [1501].log_data[3].valid := 1, [1501].log_data[4].valid := 1, [1501].time.Year := 2022, [1501].time.Month := 4, [1501].time.Day := 29, [1501].time.Hour := 2, [1501].time.Minute := 39, [1501].time.Second := 59, [1501].time.DST_ON := 1, [1502].log_data[0].min := 1.0, [1502].log_data[0].max := 1.0, [1502].log_data[0].total := 300.0, [1502].log_data[0].time := 300.0, [1502].log_data[0].minminute := 40, [1502].log_data[0].maxminute := 40, [1502].log_data[0].valid := 1, [1502].log_data[1].valid := 1, [1502].log_data[2].valid := 1, [1502].log_data[3].valid := 1, [1502].log_data[4].valid := 1, [1502].time.Year := 2022, [1502].time.Month := 4, [1502].time.Day := 29, [1502].time.Hour := 2, [1502].time.Minute := 44, [1502].time.Second := 59, [1502].time.DST_ON := 1, [1503].log_data[0].min := 1.0, [1503].log_data[0].max := 1.0, [1503].log_data[0].total := 300.0, [1503].log_data[0].time := 300.0, [1503].log_data[0].minminute := 45, [1503].log_data[0].maxminute := 45, [1503].log_data[0].valid := 1, [1503].log_data[1].valid := 1, [1503].log_data[2].valid := 1, [1503].log_data[3].valid := 1, [1503].log_data[4].valid := 1, [1503].time.Year := 2022, [1503].time.Month := 4, [1503].time.Day := 29, [1503].time.Hour := 2, [1503].time.Minute := 49, [1503].time.Second := 59, [1503].time.DST_ON := 1, [1504].log_data[0].min := 1.0, [1504].log_data[0].max := 1.0, [1504].log_data[0].total := 300.0, [1504].log_data[0].time := 300.0, [1504].log_data[0].minminute := 50,
        [1504].log_data[0].maxminute := 50, [1504].log_data[0].valid := 1, [1504].log_data[1].valid := 1, [1504].log_data[2].valid := 1, [1504].log_data[3].valid := 1, [1504].log_data[4].valid := 1, [1504].time.Year := 2022, [1504].time.Month := 4, [1504].time.Day := 29, [1504].time.Hour := 2, [1504].time.Minute := 54, [1504].time.Second := 59, [1504].time.DST_ON := 1, [1505].log_data[0].min := 1.0, [1505].log_data[0].max := 1.0, [1505].log_data[0].total := 300.0, [1505].log_data[0].time := 300.0, [1505].log_data[0].minminute := 55, [1505].log_data[0].maxminute := 55, [1505].log_data[0].valid := 1, [1505].log_data[1].valid := 1, [1505].log_data[2].valid := 1, [1505].log_data[3].valid := 1, [1505].log_data[4].valid := 1, [1505].time.Year := 2022, [1505].time.Month := 4, [1505].time.Day := 29, [1505].time.Hour := 2, [1505].time.Minute := 59, [1505].time.Second := 59, [1505].time.DST_ON := 1, [1506].log_data[0].min := 1.0, [1506].log_data[0].max := 1.0, [1506].log_data[0].total := 300.0, [1506].log_data[0].time := 300.0, [1506].log_data[0].valid := 1, [1506].log_data[1].valid := 1, [1506].log_data[2].valid := 1, [1506].log_data[3].valid := 1, [1506].log_data[4].valid := 1, [1506].time.Year := 2022, [1506].time.Month := 4, [1506].time.Day := 29, [1506].time.Hour := 3, [1506].time.Minute := 4, [1506].time.Second := 59, [1506].time.DST_ON := 1, [1507].log_data[0].min := 1.0, [1507].log_data[0].max := 1.0, [1507].log_data[0].total := 300.0, [1507].log_data[0].time := 300.0, [1507].log_data[0].minminute := 5, [1507].log_data[0].maxminute := 5, [1507].log_data[0].valid := 1, [1507].log_data[1].valid := 1, [1507].log_data[2].valid := 1, [1507].log_data[3].valid := 1, [1507].log_data[4].valid := 1, [1507].time.Year := 2022, [1507].time.Month := 4,
        [1507].time.Day := 29, [1507].time.Hour := 3, [1507].time.Minute := 9, [1507].time.Second := 59, [1507].time.DST_ON := 1, [1508].log_data[0].min := 1.0, [1508].log_data[0].max := 1.0, [1508].log_data[0].total := 300.0, [1508].log_data[0].time := 300.0, [1508].log_data[0].minminute := 10, [1508].log_data[0].maxminute := 10, [1508].log_data[0].valid := 1, [1508].log_data[1].valid := 1, [1508].log_data[2].valid := 1, [1508].log_data[3].valid := 1, [1508].log_data[4].valid := 1, [1508].time.Year := 2022, [1508].time.Month := 4, [1508].time.Day := 29, [1508].time.Hour := 3, [1508].time.Minute := 14, [1508].time.Second := 59, [1508].time.DST_ON := 1, [1509].log_data[0].min := 1.0, [1509].log_data[0].max := 1.0, [1509].log_data[0].total := 300.0, [1509].log_data[0].time := 300.0, [1509].log_data[0].minminute := 15, [1509].log_data[0].maxminute := 15, [1509].log_data[0].valid := 1, [1509].log_data[1].valid := 1, [1509].log_data[2].valid := 1, [1509].log_data[3].valid := 1, [1509].log_data[4].valid := 1, [1509].time.Year := 2022, [1509].time.Month := 4, [1509].time.Day := 29, [1509].time.Hour := 3, [1509].time.Minute := 19, [1509].time.Second := 59, [1509].time.DST_ON := 1, [1510].log_data[0].min := 1.0, [1510].log_data[0].max := 1.0, [1510].log_data[0].total := 300.0, [1510].log_data[0].time := 300.0, [1510].log_data[0].minminute := 20, [1510].log_data[0].maxminute := 20, [1510].log_data[0].valid := 1, [1510].log_data[1].valid := 1, [1510].log_data[2].valid := 1, [1510].log_data[3].valid := 1, [1510].log_data[4].valid := 1, [1510].time.Year := 2022, [1510].time.Month := 4, [1510].time.Day := 29, [1510].time.Hour := 3, [1510].time.Minute := 24, [1510].time.Second := 59, [1510].time.DST_ON := 1, [1511].log_data[0].min := 1.0,
        [1511].log_data[0].max := 1.0, [1511].log_data[0].total := 300.0, [1511].log_data[0].time := 300.0, [1511].log_data[0].minminute := 25, [1511].log_data[0].maxminute := 25, [1511].log_data[0].valid := 1, [1511].log_data[1].valid := 1, [1511].log_data[2].valid := 1, [1511].log_data[3].valid := 1, [1511].log_data[4].valid := 1, [1511].time.Year := 2022, [1511].time.Month := 4, [1511].time.Day := 29, [1511].time.Hour := 3, [1511].time.Minute := 29, [1511].time.Second := 59, [1511].time.DST_ON := 1, [1512].log_data[0].min := 1.0, [1512].log_data[0].max := 1.0, [1512].log_data[0].total := 300.0, [1512].log_data[0].time := 300.0, [1512].log_data[0].minminute := 30, [1512].log_data[0].maxminute := 30, [1512].log_data[0].valid := 1, [1512].log_data[1].valid := 1, [1512].log_data[2].valid := 1, [1512].log_data[3].valid := 1, [1512].log_data[4].valid := 1, [1512].time.Year := 2022, [1512].time.Month := 4, [1512].time.Day := 29, [1512].time.Hour := 3, [1512].time.Minute := 34, [1512].time.Second := 59, [1512].time.DST_ON := 1, [1513].log_data[0].min := 1.0, [1513].log_data[0].max := 1.0, [1513].log_data[0].total := 300.0, [1513].log_data[0].time := 300.0, [1513].log_data[0].minminute := 35, [1513].log_data[0].maxminute := 35, [1513].log_data[0].valid := 1, [1513].log_data[1].valid := 1, [1513].log_data[2].valid := 1, [1513].log_data[3].valid := 1, [1513].log_data[4].valid := 1, [1513].time.Year := 2022, [1513].time.Month := 4, [1513].time.Day := 29, [1513].time.Hour := 3, [1513].time.Minute := 39, [1513].time.Second := 59, [1513].time.DST_ON := 1, [1514].log_data[0].min := 1.0, [1514].log_data[0].max := 1.0, [1514].log_data[0].total := 300.0, [1514].log_data[0].time := 300.0, [1514].log_data[0].minminute := 40, [1514].log_data[0].maxminute := 40, [1514].log_data[0].valid := 1,
        [1514].log_data[1].valid := 1, [1514].log_data[2].valid := 1, [1514].log_data[3].valid := 1, [1514].log_data[4].valid := 1, [1514].time.Year := 2022, [1514].time.Month := 4, [1514].time.Day := 29, [1514].time.Hour := 3, [1514].time.Minute := 44, [1514].time.Second := 59, [1514].time.DST_ON := 1, [1515].log_data[0].min := 1.0, [1515].log_data[0].max := 1.0, [1515].log_data[0].total := 300.0, [1515].log_data[0].time := 300.0, [1515].log_data[0].minminute := 45, [1515].log_data[0].maxminute := 45, [1515].log_data[0].valid := 1, [1515].log_data[1].valid := 1, [1515].log_data[2].valid := 1, [1515].log_data[3].valid := 1, [1515].log_data[4].valid := 1, [1515].time.Year := 2022, [1515].time.Month := 4, [1515].time.Day := 29, [1515].time.Hour := 3, [1515].time.Minute := 49, [1515].time.Second := 59, [1515].time.DST_ON := 1, [1516].log_data[0].min := 1.0, [1516].log_data[0].max := 1.0, [1516].log_data[0].total := 300.0, [1516].log_data[0].time := 300.0, [1516].log_data[0].minminute := 50, [1516].log_data[0].maxminute := 50, [1516].log_data[0].valid := 1, [1516].log_data[1].valid := 1, [1516].log_data[2].valid := 1, [1516].log_data[3].valid := 1, [1516].log_data[4].valid := 1, [1516].time.Year := 2022, [1516].time.Month := 4, [1516].time.Day := 29, [1516].time.Hour := 3, [1516].time.Minute := 54, [1516].time.Second := 59, [1516].time.DST_ON := 1, [1517].log_data[0].min := 1.0, [1517].log_data[0].max := 1.0, [1517].log_data[0].total := 300.0, [1517].log_data[0].time := 300.0, [1517].log_data[0].minminute := 55, [1517].log_data[0].maxminute := 55, [1517].log_data[0].valid := 1, [1517].log_data[1].valid := 1, [1517].log_data[2].valid := 1, [1517].log_data[3].valid := 1, [1517].log_data[4].valid := 1, [1517].time.Year := 2022, [1517].time.Month := 4,
        [1517].time.Day := 29, [1517].time.Hour := 3, [1517].time.Minute := 59, [1517].time.Second := 59, [1517].time.DST_ON := 1, [1518].log_data[0].min := 1.0, [1518].log_data[0].max := 1.0, [1518].log_data[0].total := 300.0, [1518].log_data[0].time := 300.0, [1518].log_data[0].valid := 1, [1518].log_data[1].valid := 1, [1518].log_data[2].valid := 1, [1518].log_data[3].valid := 1, [1518].log_data[4].valid := 1, [1518].time.Year := 2022, [1518].time.Month := 4, [1518].time.Day := 29, [1518].time.Hour := 4, [1518].time.Minute := 4, [1518].time.Second := 59, [1518].time.DST_ON := 1, [1519].log_data[0].min := 1.0, [1519].log_data[0].max := 1.0, [1519].log_data[0].total := 300.0, [1519].log_data[0].time := 300.0, [1519].log_data[0].minminute := 5, [1519].log_data[0].maxminute := 5, [1519].log_data[0].valid := 1, [1519].log_data[1].valid := 1, [1519].log_data[2].valid := 1, [1519].log_data[3].valid := 1, [1519].log_data[4].valid := 1, [1519].time.Year := 2022, [1519].time.Month := 4, [1519].time.Day := 29, [1519].time.Hour := 4, [1519].time.Minute := 9, [1519].time.Second := 59, [1519].time.DST_ON := 1, [1520].log_data[0].min := 1.0, [1520].log_data[0].max := 1.0, [1520].log_data[0].total := 300.0, [1520].log_data[0].time := 300.0, [1520].log_data[0].minminute := 10, [1520].log_data[0].maxminute := 10, [1520].log_data[0].valid := 1, [1520].log_data[1].valid := 1, [1520].log_data[2].valid := 1, [1520].log_data[3].valid := 1, [1520].log_data[4].valid := 1, [1520].time.Year := 2022, [1520].time.Month := 4, [1520].time.Day := 29, [1520].time.Hour := 4, [1520].time.Minute := 14, [1520].time.Second := 59, [1520].time.DST_ON := 1, [1521].log_data[0].min := 1.0, [1521].log_data[0].max := 1.0, [1521].log_data[0].total := 300.0,
        [1521].log_data[0].time := 300.0, [1521].log_data[0].minminute := 15, [1521].log_data[0].maxminute := 15, [1521].log_data[0].valid := 1, [1521].log_data[1].valid := 1, [1521].log_data[2].valid := 1, [1521].log_data[3].valid := 1, [1521].log_data[4].valid := 1, [1521].time.Year := 2022, [1521].time.Month := 4, [1521].time.Day := 29, [1521].time.Hour := 4, [1521].time.Minute := 19, [1521].time.Second := 59, [1521].time.DST_ON := 1, [1522].log_data[0].min := 1.0, [1522].log_data[0].max := 1.0, [1522].log_data[0].total := 300.0, [1522].log_data[0].time := 300.0, [1522].log_data[0].minminute := 20, [1522].log_data[0].maxminute := 20, [1522].log_data[0].valid := 1, [1522].log_data[1].valid := 1, [1522].log_data[2].valid := 1, [1522].log_data[3].valid := 1, [1522].log_data[4].valid := 1, [1522].time.Year := 2022, [1522].time.Month := 4, [1522].time.Day := 29, [1522].time.Hour := 4, [1522].time.Minute := 24, [1522].time.Second := 59, [1522].time.DST_ON := 1, [1523].log_data[0].min := 1.0, [1523].log_data[0].max := 1.0, [1523].log_data[0].total := 300.0, [1523].log_data[0].time := 300.0, [1523].log_data[0].minminute := 25, [1523].log_data[0].maxminute := 25, [1523].log_data[0].valid := 1, [1523].log_data[1].valid := 1, [1523].log_data[2].valid := 1, [1523].log_data[3].valid := 1, [1523].log_data[4].valid := 1, [1523].time.Year := 2022, [1523].time.Month := 4, [1523].time.Day := 29, [1523].time.Hour := 4, [1523].time.Minute := 29, [1523].time.Second := 59, [1523].time.DST_ON := 1, [1524].log_data[0].min := 1.0, [1524].log_data[0].max := 1.0, [1524].log_data[0].total := 300.0, [1524].log_data[0].time := 300.0, [1524].log_data[0].minminute := 30, [1524].log_data[0].maxminute := 30, [1524].log_data[0].valid := 1, [1524].log_data[1].valid := 1, [1524].log_data[2].valid := 1,
        [1524].log_data[3].valid := 1, [1524].log_data[4].valid := 1, [1524].time.Year := 2022, [1524].time.Month := 4, [1524].time.Day := 29, [1524].time.Hour := 4, [1524].time.Minute := 34, [1524].time.Second := 59, [1524].time.DST_ON := 1, [1525].log_data[0].min := 1.0, [1525].log_data[0].max := 1.0, [1525].log_data[0].total := 300.0, [1525].log_data[0].time := 300.0, [1525].log_data[0].minminute := 35, [1525].log_data[0].maxminute := 35, [1525].log_data[0].valid := 1, [1525].log_data[1].valid := 1, [1525].log_data[2].valid := 1, [1525].log_data[3].valid := 1, [1525].log_data[4].valid := 1, [1525].time.Year := 2022, [1525].time.Month := 4, [1525].time.Day := 29, [1525].time.Hour := 4, [1525].time.Minute := 39, [1525].time.Second := 59, [1525].time.DST_ON := 1, [1526].log_data[0].min := 1.0, [1526].log_data[0].max := 1.0, [1526].log_data[0].total := 300.0, [1526].log_data[0].time := 300.0, [1526].log_data[0].minminute := 40, [1526].log_data[0].maxminute := 40, [1526].log_data[0].valid := 1, [1526].log_data[1].valid := 1, [1526].log_data[2].valid := 1, [1526].log_data[3].valid := 1, [1526].log_data[4].valid := 1, [1526].time.Year := 2022, [1526].time.Month := 4, [1526].time.Day := 29, [1526].time.Hour := 4, [1526].time.Minute := 44, [1526].time.Second := 59, [1526].time.DST_ON := 1, [1527].log_data[0].min := 1.0, [1527].log_data[0].max := 1.0, [1527].log_data[0].total := 300.0, [1527].log_data[0].time := 300.0, [1527].log_data[0].minminute := 45, [1527].log_data[0].maxminute := 45, [1527].log_data[0].valid := 1, [1527].log_data[1].valid := 1, [1527].log_data[2].valid := 1, [1527].log_data[3].valid := 1, [1527].log_data[4].valid := 1, [1527].time.Year := 2022, [1527].time.Month := 4, [1527].time.Day := 29, [1527].time.Hour := 4,
        [1527].time.Minute := 49, [1527].time.Second := 59, [1527].time.DST_ON := 1, [1528].log_data[0].min := 1.0, [1528].log_data[0].max := 1.0, [1528].log_data[0].total := 300.0, [1528].log_data[0].time := 300.0, [1528].log_data[0].minminute := 50, [1528].log_data[0].maxminute := 50, [1528].log_data[0].valid := 1, [1528].log_data[1].valid := 1, [1528].log_data[2].valid := 1, [1528].log_data[3].valid := 1, [1528].log_data[4].valid := 1, [1528].time.Year := 2022, [1528].time.Month := 4, [1528].time.Day := 29, [1528].time.Hour := 4, [1528].time.Minute := 54, [1528].time.Second := 59, [1528].time.DST_ON := 1, [1529].log_data[0].min := 1.0, [1529].log_data[0].max := 1.0, [1529].log_data[0].total := 300.0, [1529].log_data[0].time := 300.0, [1529].log_data[0].minminute := 55, [1529].log_data[0].maxminute := 55, [1529].log_data[0].valid := 1, [1529].log_data[1].valid := 1, [1529].log_data[2].valid := 1, [1529].log_data[3].valid := 1, [1529].log_data[4].valid := 1, [1529].time.Year := 2022, [1529].time.Month := 4, [1529].time.Day := 29, [1529].time.Hour := 4, [1529].time.Minute := 59, [1529].time.Second := 59, [1529].time.DST_ON := 1, [1530].log_data[0].min := 1.0, [1530].log_data[0].max := 1.0, [1530].log_data[0].total := 300.0, [1530].log_data[0].time := 300.0, [1530].log_data[0].valid := 1, [1530].log_data[1].valid := 1, [1530].log_data[2].valid := 1, [1530].log_data[3].valid := 1, [1530].log_data[4].valid := 1, [1530].time.Year := 2022, [1530].time.Month := 4, [1530].time.Day := 29, [1530].time.Hour := 5, [1530].time.Minute := 4, [1530].time.Second := 59, [1530].time.DST_ON := 1, [1531].log_data[0].min := 1.0, [1531].log_data[0].max := 1.0, [1531].log_data[0].total := 300.0, [1531].log_data[0].time := 300.0, [1531].log_data[0].minminute := 5,
        [1531].log_data[0].maxminute := 5, [1531].log_data[0].valid := 1, [1531].log_data[1].valid := 1, [1531].log_data[2].valid := 1, [1531].log_data[3].valid := 1, [1531].log_data[4].valid := 1, [1531].time.Year := 2022, [1531].time.Month := 4, [1531].time.Day := 29, [1531].time.Hour := 5, [1531].time.Minute := 9, [1531].time.Second := 59, [1531].time.DST_ON := 1, [1532].log_data[0].min := 1.0, [1532].log_data[0].max := 1.0, [1532].log_data[0].total := 300.0, [1532].log_data[0].time := 300.0, [1532].log_data[0].minminute := 10, [1532].log_data[0].maxminute := 10, [1532].log_data[0].valid := 1, [1532].log_data[1].valid := 1, [1532].log_data[2].valid := 1, [1532].log_data[3].valid := 1, [1532].log_data[4].valid := 1, [1532].time.Year := 2022, [1532].time.Month := 4, [1532].time.Day := 29, [1532].time.Hour := 5, [1532].time.Minute := 14, [1532].time.Second := 59, [1532].time.DST_ON := 1, [1533].log_data[0].min := 1.0, [1533].log_data[0].max := 1.0, [1533].log_data[0].total := 300.0, [1533].log_data[0].time := 300.0, [1533].log_data[0].minminute := 15, [1533].log_data[0].maxminute := 15, [1533].log_data[0].valid := 1, [1533].log_data[1].valid := 1, [1533].log_data[2].valid := 1, [1533].log_data[3].valid := 1, [1533].log_data[4].valid := 1, [1533].time.Year := 2022, [1533].time.Month := 4, [1533].time.Day := 29, [1533].time.Hour := 5, [1533].time.Minute := 19, [1533].time.Second := 59, [1533].time.DST_ON := 1, [1534].log_data[0].min := 1.0, [1534].log_data[0].max := 1.0, [1534].log_data[0].total := 300.0, [1534].log_data[0].time := 300.0, [1534].log_data[0].minminute := 20, [1534].log_data[0].maxminute := 20, [1534].log_data[0].valid := 1, [1534].log_data[1].valid := 1, [1534].log_data[2].valid := 1, [1534].log_data[3].valid := 1, [1534].log_data[4].valid := 1,
        [1534].time.Year := 2022, [1534].time.Month := 4, [1534].time.Day := 29, [1534].time.Hour := 5, [1534].time.Minute := 24, [1534].time.Second := 59, [1534].time.DST_ON := 1, [1535].log_data[0].min := 1.0, [1535].log_data[0].max := 1.0, [1535].log_data[0].total := 300.0, [1535].log_data[0].time := 300.0, [1535].log_data[0].minminute := 25, [1535].log_data[0].maxminute := 25, [1535].log_data[0].valid := 1, [1535].log_data[1].valid := 1, [1535].log_data[2].valid := 1, [1535].log_data[3].valid := 1, [1535].log_data[4].valid := 1, [1535].time.Year := 2022, [1535].time.Month := 4, [1535].time.Day := 29, [1535].time.Hour := 5, [1535].time.Minute := 29, [1535].time.Second := 59, [1535].time.DST_ON := 1, [1536].log_data[0].min := 1.0, [1536].log_data[0].max := 1.0, [1536].log_data[0].total := 300.0, [1536].log_data[0].time := 300.0, [1536].log_data[0].minminute := 30, [1536].log_data[0].maxminute := 30, [1536].log_data[0].valid := 1, [1536].log_data[1].valid := 1, [1536].log_data[2].valid := 1, [1536].log_data[3].valid := 1, [1536].log_data[4].valid := 1, [1536].time.Year := 2022, [1536].time.Month := 4, [1536].time.Day := 29, [1536].time.Hour := 5, [1536].time.Minute := 34, [1536].time.Second := 59, [1536].time.DST_ON := 1, [1537].log_data[0].min := 1.0, [1537].log_data[0].max := 1.0, [1537].log_data[0].total := 300.0, [1537].log_data[0].time := 300.0, [1537].log_data[0].minminute := 35, [1537].log_data[0].maxminute := 35, [1537].log_data[0].valid := 1, [1537].log_data[1].valid := 1, [1537].log_data[2].valid := 1, [1537].log_data[3].valid := 1, [1537].log_data[4].valid := 1, [1537].time.Year := 2022, [1537].time.Month := 4, [1537].time.Day := 29, [1537].time.Hour := 5, [1537].time.Minute := 39, [1537].time.Second := 59,
        [1537].time.DST_ON := 1, [1538].log_data[0].min := 1.0, [1538].log_data[0].max := 1.0, [1538].log_data[0].total := 300.0, [1538].log_data[0].time := 300.0, [1538].log_data[0].minminute := 40, [1538].log_data[0].maxminute := 40, [1538].log_data[0].valid := 1, [1538].log_data[1].valid := 1, [1538].log_data[2].valid := 1, [1538].log_data[3].valid := 1, [1538].log_data[4].valid := 1, [1538].time.Year := 2022, [1538].time.Month := 4, [1538].time.Day := 29, [1538].time.Hour := 5, [1538].time.Minute := 44, [1538].time.Second := 59, [1538].time.DST_ON := 1, [1539].log_data[0].min := 1.0, [1539].log_data[0].max := 1.0, [1539].log_data[0].total := 300.0, [1539].log_data[0].time := 300.0, [1539].log_data[0].minminute := 45, [1539].log_data[0].maxminute := 45, [1539].log_data[0].valid := 1, [1539].log_data[1].valid := 1, [1539].log_data[2].valid := 1, [1539].log_data[3].valid := 1, [1539].log_data[4].valid := 1, [1539].time.Year := 2022, [1539].time.Month := 4, [1539].time.Day := 29, [1539].time.Hour := 5, [1539].time.Minute := 49, [1539].time.Second := 59, [1539].time.DST_ON := 1, [1540].log_data[0].min := 1.0, [1540].log_data[0].max := 1.0, [1540].log_data[0].total := 300.0, [1540].log_data[0].time := 300.0, [1540].log_data[0].minminute := 50, [1540].log_data[0].maxminute := 50, [1540].log_data[0].valid := 1, [1540].log_data[1].valid := 1, [1540].log_data[2].valid := 1, [1540].log_data[3].valid := 1, [1540].log_data[4].valid := 1, [1540].time.Year := 2022, [1540].time.Month := 4, [1540].time.Day := 29, [1540].time.Hour := 5, [1540].time.Minute := 54, [1540].time.Second := 59, [1540].time.DST_ON := 1, [1541].log_data[0].min := 1.0, [1541].log_data[0].max := 1.0, [1541].log_data[0].total := 300.0, [1541].log_data[0].time := 300.0, [1541].log_data[0].minminute := 55,
        [1541].log_data[0].maxminute := 55, [1541].log_data[0].valid := 1, [1541].log_data[1].valid := 1, [1541].log_data[2].valid := 1, [1541].log_data[3].valid := 1, [1541].log_data[4].valid := 1, [1541].time.Year := 2022, [1541].time.Month := 4, [1541].time.Day := 29, [1541].time.Hour := 5, [1541].time.Minute := 59, [1541].time.Second := 59, [1541].time.DST_ON := 1, [1542].log_data[0].min := 1.0, [1542].log_data[0].max := 1.0, [1542].log_data[0].total := 300.0, [1542].log_data[0].time := 300.0, [1542].log_data[0].valid := 1, [1542].log_data[1].valid := 1, [1542].log_data[2].valid := 1, [1542].log_data[3].valid := 1, [1542].log_data[4].valid := 1, [1542].time.Year := 2022, [1542].time.Month := 4, [1542].time.Day := 29, [1542].time.Hour := 6, [1542].time.Minute := 4, [1542].time.Second := 59, [1542].time.DST_ON := 1, [1543].log_data[0].min := 1.0, [1543].log_data[0].max := 1.0, [1543].log_data[0].total := 300.0, [1543].log_data[0].time := 300.0, [1543].log_data[0].minminute := 5, [1543].log_data[0].maxminute := 5, [1543].log_data[0].valid := 1, [1543].log_data[1].valid := 1, [1543].log_data[2].valid := 1, [1543].log_data[3].valid := 1, [1543].log_data[4].valid := 1, [1543].time.Year := 2022, [1543].time.Month := 4, [1543].time.Day := 29, [1543].time.Hour := 6, [1543].time.Minute := 9, [1543].time.Second := 59, [1543].time.DST_ON := 1, [1544].log_data[0].min := 1.0, [1544].log_data[0].max := 1.0, [1544].log_data[0].total := 300.0, [1544].log_data[0].time := 300.0, [1544].log_data[0].minminute := 10, [1544].log_data[0].maxminute := 10, [1544].log_data[0].valid := 1, [1544].log_data[1].valid := 1, [1544].log_data[2].valid := 1, [1544].log_data[3].valid := 1, [1544].log_data[4].valid := 1, [1544].time.Year := 2022, [1544].time.Month := 4,
        [1544].time.Day := 29, [1544].time.Hour := 6, [1544].time.Minute := 14, [1544].time.Second := 59, [1544].time.DST_ON := 1, [1545].log_data[0].min := 1.0, [1545].log_data[0].max := 1.0, [1545].log_data[0].total := 299.999, [1545].log_data[0].time := 299.999, [1545].log_data[0].minminute := 15, [1545].log_data[0].maxminute := 15, [1545].log_data[0].valid := 1, [1545].log_data[1].valid := 1, [1545].log_data[2].valid := 1, [1545].log_data[3].valid := 1, [1545].log_data[4].valid := 1, [1545].time.Year := 2022, [1545].time.Month := 4, [1545].time.Day := 29, [1545].time.Hour := 6, [1545].time.Minute := 19, [1545].time.Second := 59, [1545].time.DST_ON := 1, [1546].log_data[0].min := 1.0, [1546].log_data[0].max := 1.0, [1546].log_data[0].total := 300.0, [1546].log_data[0].time := 300.0, [1546].log_data[0].minminute := 20, [1546].log_data[0].maxminute := 20, [1546].log_data[0].valid := 1, [1546].log_data[1].valid := 1, [1546].log_data[2].valid := 1, [1546].log_data[3].valid := 1, [1546].log_data[4].valid := 1, [1546].time.Year := 2022, [1546].time.Month := 4, [1546].time.Day := 29, [1546].time.Hour := 6, [1546].time.Minute := 24, [1546].time.Second := 59, [1546].time.DST_ON := 1, [1547].log_data[0].min := 1.0, [1547].log_data[0].max := 1.0, [1547].log_data[0].total := 300.0, [1547].log_data[0].time := 300.0, [1547].log_data[0].minminute := 25, [1547].log_data[0].maxminute := 25, [1547].log_data[0].valid := 1, [1547].log_data[1].valid := 1, [1547].log_data[2].valid := 1, [1547].log_data[3].valid := 1, [1547].log_data[4].valid := 1, [1547].time.Year := 2022, [1547].time.Month := 4, [1547].time.Day := 29, [1547].time.Hour := 6, [1547].time.Minute := 29, [1547].time.Second := 59, [1547].time.DST_ON := 1, [1548].log_data[0].min := 1.0,
        [1548].log_data[0].max := 1.0, [1548].log_data[0].total := 300.0, [1548].log_data[0].time := 300.0, [1548].log_data[0].minminute := 30, [1548].log_data[0].maxminute := 30, [1548].log_data[0].valid := 1, [1548].log_data[1].valid := 1, [1548].log_data[2].valid := 1, [1548].log_data[3].valid := 1, [1548].log_data[4].valid := 1, [1548].time.Year := 2022, [1548].time.Month := 4, [1548].time.Day := 29, [1548].time.Hour := 6, [1548].time.Minute := 34, [1548].time.Second := 59, [1548].time.DST_ON := 1, [1549].log_data[0].min := 1.0, [1549].log_data[0].max := 1.0, [1549].log_data[0].total := 300.0, [1549].log_data[0].time := 300.0, [1549].log_data[0].minminute := 35, [1549].log_data[0].maxminute := 35, [1549].log_data[0].valid := 1, [1549].log_data[1].valid := 1, [1549].log_data[2].valid := 1, [1549].log_data[3].valid := 1, [1549].log_data[4].valid := 1, [1549].time.Year := 2022, [1549].time.Month := 4, [1549].time.Day := 29, [1549].time.Hour := 6, [1549].time.Minute := 39, [1549].time.Second := 59, [1549].time.DST_ON := 1, [1550].log_data[0].min := 1.0, [1550].log_data[0].max := 1.0, [1550].log_data[0].total := 300.0, [1550].log_data[0].time := 300.0, [1550].log_data[0].minminute := 40, [1550].log_data[0].maxminute := 40, [1550].log_data[0].valid := 1, [1550].log_data[1].valid := 1, [1550].log_data[2].valid := 1, [1550].log_data[3].valid := 1, [1550].log_data[4].valid := 1, [1550].time.Year := 2022, [1550].time.Month := 4, [1550].time.Day := 29, [1550].time.Hour := 6, [1550].time.Minute := 44, [1550].time.Second := 59, [1550].time.DST_ON := 1, [1551].log_data[0].min := 1.0, [1551].log_data[0].max := 1.0, [1551].log_data[0].total := 300.0, [1551].log_data[0].time := 300.0, [1551].log_data[0].minminute := 45, [1551].log_data[0].maxminute := 45, [1551].log_data[0].valid := 1,
        [1551].log_data[1].valid := 1, [1551].log_data[2].valid := 1, [1551].log_data[3].valid := 1, [1551].log_data[4].valid := 1, [1551].time.Year := 2022, [1551].time.Month := 4, [1551].time.Day := 29, [1551].time.Hour := 6, [1551].time.Minute := 49, [1551].time.Second := 59, [1551].time.DST_ON := 1, [1552].log_data[0].min := 1.0, [1552].log_data[0].max := 1.0, [1552].log_data[0].total := 300.0, [1552].log_data[0].time := 300.0, [1552].log_data[0].minminute := 50, [1552].log_data[0].maxminute := 50, [1552].log_data[0].valid := 1, [1552].log_data[1].valid := 1, [1552].log_data[2].valid := 1, [1552].log_data[3].valid := 1, [1552].log_data[4].valid := 1, [1552].time.Year := 2022, [1552].time.Month := 4, [1552].time.Day := 29, [1552].time.Hour := 6, [1552].time.Minute := 54, [1552].time.Second := 59, [1552].time.DST_ON := 1, [1553].log_data[0].min := 1.0, [1553].log_data[0].max := 1.0, [1553].log_data[0].total := 300.0, [1553].log_data[0].time := 300.0, [1553].log_data[0].minminute := 55, [1553].log_data[0].maxminute := 55, [1553].log_data[0].valid := 1, [1553].log_data[1].valid := 1, [1553].log_data[2].valid := 1, [1553].log_data[3].valid := 1, [1553].log_data[4].valid := 1, [1553].time.Year := 2022, [1553].time.Month := 4, [1553].time.Day := 29, [1553].time.Hour := 6, [1553].time.Minute := 59, [1553].time.Second := 59, [1553].time.DST_ON := 1, [1554].log_data[0].min := 1.0, [1554].log_data[0].max := 1.0, [1554].log_data[0].total := 300.0, [1554].log_data[0].time := 300.0, [1554].log_data[0].valid := 1, [1554].log_data[1].valid := 1, [1554].log_data[2].valid := 1, [1554].log_data[3].valid := 1, [1554].log_data[4].valid := 1, [1554].time.Year := 2022, [1554].time.Month := 4, [1554].time.Day := 29, [1554].time.Hour := 7,
        [1554].time.Minute := 4, [1554].time.Second := 59, [1554].time.DST_ON := 1, [1555].log_data[0].min := 1.0, [1555].log_data[0].max := 1.0, [1555].log_data[0].total := 300.0, [1555].log_data[0].time := 300.0, [1555].log_data[0].minminute := 5, [1555].log_data[0].maxminute := 5, [1555].log_data[0].valid := 1, [1555].log_data[1].valid := 1, [1555].log_data[2].valid := 1, [1555].log_data[3].valid := 1, [1555].log_data[4].valid := 1, [1555].time.Year := 2022, [1555].time.Month := 4, [1555].time.Day := 29, [1555].time.Hour := 7, [1555].time.Minute := 9, [1555].time.Second := 59, [1555].time.DST_ON := 1, [1556].log_data[0].min := 1.0, [1556].log_data[0].max := 1.0, [1556].log_data[0].total := 300.0, [1556].log_data[0].time := 300.0, [1556].log_data[0].minminute := 10, [1556].log_data[0].maxminute := 10, [1556].log_data[0].valid := 1, [1556].log_data[1].valid := 1, [1556].log_data[2].valid := 1, [1556].log_data[3].valid := 1, [1556].log_data[4].valid := 1, [1556].time.Year := 2022, [1556].time.Month := 4, [1556].time.Day := 29, [1556].time.Hour := 7, [1556].time.Minute := 14, [1556].time.Second := 59, [1556].time.DST_ON := 1, [1557].log_data[0].min := 1.0, [1557].log_data[0].max := 1.0, [1557].log_data[0].total := 300.0, [1557].log_data[0].time := 300.0, [1557].log_data[0].minminute := 15, [1557].log_data[0].maxminute := 15, [1557].log_data[0].valid := 1, [1557].log_data[1].valid := 1, [1557].log_data[2].valid := 1, [1557].log_data[3].valid := 1, [1557].log_data[4].valid := 1, [1557].time.Year := 2022, [1557].time.Month := 4, [1557].time.Day := 29, [1557].time.Hour := 7, [1557].time.Minute := 19, [1557].time.Second := 59, [1557].time.DST_ON := 1, [1558].log_data[0].min := 1.0, [1558].log_data[0].max := 1.0, [1558].log_data[0].total := 300.0,
        [1558].log_data[0].time := 300.0, [1558].log_data[0].minminute := 20, [1558].log_data[0].maxminute := 20, [1558].log_data[0].valid := 1, [1558].log_data[1].valid := 1, [1558].log_data[2].valid := 1, [1558].log_data[3].valid := 1, [1558].log_data[4].valid := 1, [1558].time.Year := 2022, [1558].time.Month := 4, [1558].time.Day := 29, [1558].time.Hour := 7, [1558].time.Minute := 24, [1558].time.Second := 59, [1558].time.DST_ON := 1, [1559].log_data[0].min := 1.0, [1559].log_data[0].max := 1.0, [1559].log_data[0].total := 300.0, [1559].log_data[0].time := 300.0, [1559].log_data[0].minminute := 25, [1559].log_data[0].maxminute := 25, [1559].log_data[0].valid := 1, [1559].log_data[1].valid := 1, [1559].log_data[2].valid := 1, [1559].log_data[3].valid := 1, [1559].log_data[4].valid := 1, [1559].time.Year := 2022, [1559].time.Month := 4, [1559].time.Day := 29, [1559].time.Hour := 7, [1559].time.Minute := 29, [1559].time.Second := 59, [1559].time.DST_ON := 1, [1560].log_data[0].min := 1.0, [1560].log_data[0].max := 1.0, [1560].log_data[0].total := 300.0, [1560].log_data[0].time := 300.0, [1560].log_data[0].minminute := 30, [1560].log_data[0].maxminute := 30, [1560].log_data[0].valid := 1, [1560].log_data[1].valid := 1, [1560].log_data[2].valid := 1, [1560].log_data[3].valid := 1, [1560].log_data[4].valid := 1, [1560].time.Year := 2022, [1560].time.Month := 4, [1560].time.Day := 29, [1560].time.Hour := 7, [1560].time.Minute := 34, [1560].time.Second := 59, [1560].time.DST_ON := 1, [1561].log_data[0].min := 1.0, [1561].log_data[0].max := 1.0, [1561].log_data[0].total := 300.0, [1561].log_data[0].time := 300.0, [1561].log_data[0].minminute := 35, [1561].log_data[0].maxminute := 35, [1561].log_data[0].valid := 1, [1561].log_data[1].valid := 1, [1561].log_data[2].valid := 1,
        [1561].log_data[3].valid := 1, [1561].log_data[4].valid := 1, [1561].time.Year := 2022, [1561].time.Month := 4, [1561].time.Day := 29, [1561].time.Hour := 7, [1561].time.Minute := 39, [1561].time.Second := 59, [1561].time.DST_ON := 1, [1562].log_data[0].min := 1.0, [1562].log_data[0].max := 1.0, [1562].log_data[0].total := 299.999, [1562].log_data[0].time := 299.999, [1562].log_data[0].minminute := 40, [1562].log_data[0].maxminute := 40, [1562].log_data[0].valid := 1, [1562].log_data[1].valid := 1, [1562].log_data[2].valid := 1, [1562].log_data[3].valid := 1, [1562].log_data[4].valid := 1, [1562].time.Year := 2022, [1562].time.Month := 4, [1562].time.Day := 29, [1562].time.Hour := 7, [1562].time.Minute := 44, [1562].time.Second := 59, [1562].time.DST_ON := 1, [1563].log_data[0].min := 1.0, [1563].log_data[0].max := 1.0, [1563].log_data[0].total := 300.0, [1563].log_data[0].time := 300.0, [1563].log_data[0].minminute := 45, [1563].log_data[0].maxminute := 45, [1563].log_data[0].valid := 1, [1563].log_data[1].valid := 1, [1563].log_data[2].valid := 1, [1563].log_data[3].valid := 1, [1563].log_data[4].valid := 1, [1563].time.Year := 2022, [1563].time.Month := 4, [1563].time.Day := 29, [1563].time.Hour := 7, [1563].time.Minute := 49, [1563].time.Second := 59, [1563].time.DST_ON := 1, [1564].log_data[0].min := 1.0, [1564].log_data[0].max := 1.0, [1564].log_data[0].total := 300.0, [1564].log_data[0].time := 300.0, [1564].log_data[0].minminute := 50, [1564].log_data[0].maxminute := 50, [1564].log_data[0].valid := 1, [1564].log_data[1].valid := 1, [1564].log_data[2].valid := 1, [1564].log_data[3].valid := 1, [1564].log_data[4].valid := 1, [1564].time.Year := 2022, [1564].time.Month := 4, [1564].time.Day := 29, [1564].time.Hour := 7,
        [1564].time.Minute := 54, [1564].time.Second := 59, [1564].time.DST_ON := 1, [1565].log_data[0].min := 1.0, [1565].log_data[0].max := 1.0, [1565].log_data[0].total := 300.0, [1565].log_data[0].time := 300.0, [1565].log_data[0].minminute := 55, [1565].log_data[0].maxminute := 55, [1565].log_data[0].valid := 1, [1565].log_data[1].valid := 1, [1565].log_data[2].valid := 1, [1565].log_data[3].valid := 1, [1565].log_data[4].valid := 1, [1565].time.Year := 2022, [1565].time.Month := 4, [1565].time.Day := 29, [1565].time.Hour := 7, [1565].time.Minute := 59, [1565].time.Second := 59, [1565].time.DST_ON := 1, [1566].log_data[0].min := 1.0, [1566].log_data[0].max := 1.0, [1566].log_data[0].total := 300.0, [1566].log_data[0].time := 300.0, [1566].log_data[0].valid := 1, [1566].log_data[1].valid := 1, [1566].log_data[2].valid := 1, [1566].log_data[3].valid := 1, [1566].log_data[4].valid := 1, [1566].time.Year := 2022, [1566].time.Month := 4, [1566].time.Day := 29, [1566].time.Hour := 8, [1566].time.Minute := 4, [1566].time.Second := 59, [1566].time.DST_ON := 1, [1567].log_data[0].min := 1.0, [1567].log_data[0].max := 1.0, [1567].log_data[0].total := 300.0, [1567].log_data[0].time := 300.0, [1567].log_data[0].minminute := 5, [1567].log_data[0].maxminute := 5, [1567].log_data[0].valid := 1, [1567].log_data[1].valid := 1, [1567].log_data[2].valid := 1, [1567].log_data[3].valid := 1, [1567].log_data[4].valid := 1, [1567].time.Year := 2022, [1567].time.Month := 4, [1567].time.Day := 29, [1567].time.Hour := 8, [1567].time.Minute := 9, [1567].time.Second := 59, [1567].time.DST_ON := 1, [1568].log_data[0].min := 1.0, [1568].log_data[0].max := 1.0, [1568].log_data[0].total := 300.0, [1568].log_data[0].time := 300.0, [1568].log_data[0].minminute := 10,
        [1568].log_data[0].maxminute := 10, [1568].log_data[0].valid := 1, [1568].log_data[1].valid := 1, [1568].log_data[2].valid := 1, [1568].log_data[3].valid := 1, [1568].log_data[4].valid := 1, [1568].time.Year := 2022, [1568].time.Month := 4, [1568].time.Day := 29, [1568].time.Hour := 8, [1568].time.Minute := 14, [1568].time.Second := 59, [1568].time.DST_ON := 1, [1569].log_data[0].min := 1.0, [1569].log_data[0].max := 1.0, [1569].log_data[0].total := 300.0, [1569].log_data[0].time := 300.0, [1569].log_data[0].minminute := 15, [1569].log_data[0].maxminute := 15, [1569].log_data[0].valid := 1, [1569].log_data[1].valid := 1, [1569].log_data[2].valid := 1, [1569].log_data[3].valid := 1, [1569].log_data[4].valid := 1, [1569].time.Year := 2022, [1569].time.Month := 4, [1569].time.Day := 29, [1569].time.Hour := 8, [1569].time.Minute := 19, [1569].time.Second := 59, [1569].time.DST_ON := 1, [1570].log_data[0].min := 1.0, [1570].log_data[0].max := 1.0, [1570].log_data[0].total := 300.0, [1570].log_data[0].time := 300.0, [1570].log_data[0].minminute := 20, [1570].log_data[0].maxminute := 20, [1570].log_data[0].valid := 1, [1570].log_data[1].valid := 1, [1570].log_data[2].valid := 1, [1570].log_data[3].valid := 1, [1570].log_data[4].valid := 1, [1570].time.Year := 2022, [1570].time.Month := 4, [1570].time.Day := 29, [1570].time.Hour := 8, [1570].time.Minute := 24, [1570].time.Second := 59, [1570].time.DST_ON := 1, [1571].log_data[0].min := 1.0, [1571].log_data[0].max := 1.0, [1571].log_data[0].total := 300.0, [1571].log_data[0].time := 300.0, [1571].log_data[0].minminute := 25, [1571].log_data[0].maxminute := 25, [1571].log_data[0].valid := 1, [1571].log_data[1].valid := 1, [1571].log_data[2].valid := 1, [1571].log_data[3].valid := 1, [1571].log_data[4].valid := 1,
        [1571].time.Year := 2022, [1571].time.Month := 4, [1571].time.Day := 29, [1571].time.Hour := 8, [1571].time.Minute := 29, [1571].time.Second := 59, [1571].time.DST_ON := 1, [1572].log_data[0].min := 1.0, [1572].log_data[0].max := 1.0, [1572].log_data[0].total := 300.0, [1572].log_data[0].time := 300.0, [1572].log_data[0].minminute := 30, [1572].log_data[0].maxminute := 30, [1572].log_data[0].valid := 1, [1572].log_data[1].valid := 1, [1572].log_data[2].valid := 1, [1572].log_data[3].valid := 1, [1572].log_data[4].valid := 1, [1572].time.Year := 2022, [1572].time.Month := 4, [1572].time.Day := 29, [1572].time.Hour := 8, [1572].time.Minute := 34, [1572].time.Second := 59, [1572].time.DST_ON := 1, [1573].log_data[0].min := 1.0, [1573].log_data[0].max := 1.0, [1573].log_data[0].total := 300.0, [1573].log_data[0].time := 300.0, [1573].log_data[0].minminute := 35, [1573].log_data[0].maxminute := 35, [1573].log_data[0].valid := 1, [1573].log_data[1].valid := 1, [1573].log_data[2].valid := 1, [1573].log_data[3].valid := 1, [1573].log_data[4].valid := 1, [1573].time.Year := 2022, [1573].time.Month := 4, [1573].time.Day := 29, [1573].time.Hour := 8, [1573].time.Minute := 39, [1573].time.Second := 59, [1573].time.DST_ON := 1, [1574].log_data[0].min := 1.0, [1574].log_data[0].max := 1.0, [1574].log_data[0].total := 300.0, [1574].log_data[0].time := 300.0, [1574].log_data[0].minminute := 40, [1574].log_data[0].maxminute := 40, [1574].log_data[0].valid := 1, [1574].log_data[1].valid := 1, [1574].log_data[2].valid := 1, [1574].log_data[3].valid := 1, [1574].log_data[4].valid := 1, [1574].time.Year := 2022, [1574].time.Month := 4, [1574].time.Day := 29, [1574].time.Hour := 8, [1574].time.Minute := 44, [1574].time.Second := 59,
        [1574].time.DST_ON := 1, [1575].log_data[0].min := 1.0, [1575].log_data[0].max := 1.0, [1575].log_data[0].total := 300.0, [1575].log_data[0].time := 300.0, [1575].log_data[0].minminute := 45, [1575].log_data[0].maxminute := 45, [1575].log_data[0].valid := 1, [1575].log_data[1].valid := 1, [1575].log_data[2].valid := 1, [1575].log_data[3].valid := 1, [1575].log_data[4].valid := 1, [1575].time.Year := 2022, [1575].time.Month := 4, [1575].time.Day := 29, [1575].time.Hour := 8, [1575].time.Minute := 49, [1575].time.Second := 59, [1575].time.DST_ON := 1, [1576].log_data[0].min := 1.0, [1576].log_data[0].max := 1.0, [1576].log_data[0].total := 300.0, [1576].log_data[0].time := 300.0, [1576].log_data[0].minminute := 50, [1576].log_data[0].maxminute := 50, [1576].log_data[0].valid := 1, [1576].log_data[1].valid := 1, [1576].log_data[2].valid := 1, [1576].log_data[3].valid := 1, [1576].log_data[4].valid := 1, [1576].time.Year := 2022, [1576].time.Month := 4, [1576].time.Day := 29, [1576].time.Hour := 8, [1576].time.Minute := 54, [1576].time.Second := 59, [1576].time.DST_ON := 1, [1577].log_data[0].min := 1.0, [1577].log_data[0].max := 1.0, [1577].log_data[0].total := 300.0, [1577].log_data[0].time := 300.0, [1577].log_data[0].minminute := 55, [1577].log_data[0].maxminute := 55, [1577].log_data[0].valid := 1, [1577].log_data[1].valid := 1, [1577].log_data[2].valid := 1, [1577].log_data[3].valid := 1, [1577].log_data[4].valid := 1, [1577].time.Year := 2022, [1577].time.Month := 4, [1577].time.Day := 29, [1577].time.Hour := 8, [1577].time.Minute := 59, [1577].time.Second := 59, [1577].time.DST_ON := 1, [1578].log_data[0].min := 1.0, [1578].log_data[0].max := 1.0, [1578].log_data[0].total := 300.0, [1578].log_data[0].time := 300.0, [1578].log_data[0].valid := 1,
        [1578].log_data[1].valid := 1, [1578].log_data[2].valid := 1, [1578].log_data[3].valid := 1, [1578].log_data[4].valid := 1, [1578].time.Year := 2022, [1578].time.Month := 4, [1578].time.Day := 29, [1578].time.Hour := 9, [1578].time.Minute := 4, [1578].time.Second := 59, [1578].time.DST_ON := 1, [1579].log_data[0].min := 1.0, [1579].log_data[0].max := 1.0, [1579].log_data[0].total := 300.0, [1579].log_data[0].time := 300.0, [1579].log_data[0].minminute := 5, [1579].log_data[0].maxminute := 5, [1579].log_data[0].valid := 1, [1579].log_data[1].valid := 1, [1579].log_data[2].valid := 1, [1579].log_data[3].valid := 1, [1579].log_data[4].valid := 1, [1579].time.Year := 2022, [1579].time.Month := 4, [1579].time.Day := 29, [1579].time.Hour := 9, [1579].time.Minute := 9, [1579].time.Second := 59, [1579].time.DST_ON := 1, [1580].log_data[0].min := 1.0, [1580].log_data[0].max := 1.0, [1580].log_data[0].total := 300.0, [1580].log_data[0].time := 300.0, [1580].log_data[0].minminute := 10, [1580].log_data[0].maxminute := 10, [1580].log_data[0].valid := 1, [1580].log_data[1].valid := 1, [1580].log_data[2].valid := 1, [1580].log_data[3].valid := 1, [1580].log_data[4].valid := 1, [1580].time.Year := 2022, [1580].time.Month := 4, [1580].time.Day := 29, [1580].time.Hour := 9, [1580].time.Minute := 14, [1580].time.Second := 59, [1580].time.DST_ON := 1, [1581].log_data[0].min := 1.0, [1581].log_data[0].max := 1.0, [1581].log_data[0].total := 300.0, [1581].log_data[0].time := 300.0, [1581].log_data[0].minminute := 15, [1581].log_data[0].maxminute := 15, [1581].log_data[0].valid := 1, [1581].log_data[1].valid := 1, [1581].log_data[2].valid := 1, [1581].log_data[3].valid := 1, [1581].log_data[4].valid := 1, [1581].time.Year := 2022, [1581].time.Month := 4,
        [1581].time.Day := 29, [1581].time.Hour := 9, [1581].time.Minute := 19, [1581].time.Second := 59, [1581].time.DST_ON := 1, [1582].log_data[0].min := 1.0, [1582].log_data[0].max := 1.0, [1582].log_data[0].total := 300.0, [1582].log_data[0].time := 300.0, [1582].log_data[0].minminute := 20, [1582].log_data[0].maxminute := 20, [1582].log_data[0].valid := 1, [1582].log_data[1].valid := 1, [1582].log_data[2].valid := 1, [1582].log_data[3].valid := 1, [1582].log_data[4].valid := 1, [1582].time.Year := 2022, [1582].time.Month := 4, [1582].time.Day := 29, [1582].time.Hour := 9, [1582].time.Minute := 24, [1582].time.Second := 59, [1582].time.DST_ON := 1, [1583].log_data[0].min := 1.0, [1583].log_data[0].max := 1.0, [1583].log_data[0].total := 300.0, [1583].log_data[0].time := 300.0, [1583].log_data[0].minminute := 25, [1583].log_data[0].maxminute := 25, [1583].log_data[0].valid := 1, [1583].log_data[1].valid := 1, [1583].log_data[2].valid := 1, [1583].log_data[3].valid := 1, [1583].log_data[4].valid := 1, [1583].time.Year := 2022, [1583].time.Month := 4, [1583].time.Day := 29, [1583].time.Hour := 9, [1583].time.Minute := 29, [1583].time.Second := 59, [1583].time.DST_ON := 1, [1584].log_data[0].min := 1.0, [1584].log_data[0].max := 1.0, [1584].log_data[0].total := 300.0, [1584].log_data[0].time := 300.0, [1584].log_data[0].minminute := 30, [1584].log_data[0].maxminute := 30, [1584].log_data[0].valid := 1, [1584].log_data[1].valid := 1, [1584].log_data[2].valid := 1, [1584].log_data[3].valid := 1, [1584].log_data[4].valid := 1, [1584].time.Year := 2022, [1584].time.Month := 4, [1584].time.Day := 29, [1584].time.Hour := 9, [1584].time.Minute := 34, [1584].time.Second := 59, [1584].time.DST_ON := 1, [1585].log_data[0].min := 1.0,
        [1585].log_data[0].max := 1.0, [1585].log_data[0].total := 300.0, [1585].log_data[0].time := 300.0, [1585].log_data[0].minminute := 35, [1585].log_data[0].maxminute := 35, [1585].log_data[0].valid := 1, [1585].log_data[1].valid := 1, [1585].log_data[2].valid := 1, [1585].log_data[3].valid := 1, [1585].log_data[4].valid := 1, [1585].time.Year := 2022, [1585].time.Month := 4, [1585].time.Day := 29, [1585].time.Hour := 9, [1585].time.Minute := 39, [1585].time.Second := 59, [1585].time.DST_ON := 1, [1586].log_data[0].min := 1.0, [1586].log_data[0].max := 1.0, [1586].log_data[0].total := 299.999, [1586].log_data[0].time := 299.999, [1586].log_data[0].minminute := 40, [1586].log_data[0].maxminute := 40, [1586].log_data[0].valid := 1, [1586].log_data[1].valid := 1, [1586].log_data[2].valid := 1, [1586].log_data[3].valid := 1, [1586].log_data[4].valid := 1, [1586].time.Year := 2022, [1586].time.Month := 4, [1586].time.Day := 29, [1586].time.Hour := 9, [1586].time.Minute := 44, [1586].time.Second := 59, [1586].time.DST_ON := 1, [1587].log_data[0].min := 1.0, [1587].log_data[0].max := 1.0, [1587].log_data[0].total := 300.0, [1587].log_data[0].time := 300.0, [1587].log_data[0].minminute := 45, [1587].log_data[0].maxminute := 45, [1587].log_data[0].valid := 1, [1587].log_data[1].valid := 1, [1587].log_data[2].valid := 1, [1587].log_data[3].valid := 1, [1587].log_data[4].valid := 1, [1587].time.Year := 2022, [1587].time.Month := 4, [1587].time.Day := 29, [1587].time.Hour := 9, [1587].time.Minute := 49, [1587].time.Second := 59, [1587].time.DST_ON := 1, [1588].log_data[0].min := 1.0, [1588].log_data[0].max := 1.0, [1588].log_data[0].total := 300.0, [1588].log_data[0].time := 300.0, [1588].log_data[0].minminute := 50, [1588].log_data[0].maxminute := 50, [1588].log_data[0].valid := 1,
        [1588].log_data[1].valid := 1, [1588].log_data[2].valid := 1, [1588].log_data[3].valid := 1, [1588].log_data[4].valid := 1, [1588].time.Year := 2022, [1588].time.Month := 4, [1588].time.Day := 29, [1588].time.Hour := 9, [1588].time.Minute := 54, [1588].time.Second := 59, [1588].time.DST_ON := 1, [1589].log_data[0].min := 1.0, [1589].log_data[0].max := 1.0, [1589].log_data[0].total := 300.0, [1589].log_data[0].time := 300.0, [1589].log_data[0].minminute := 55, [1589].log_data[0].maxminute := 55, [1589].log_data[0].valid := 1, [1589].log_data[1].valid := 1, [1589].log_data[2].valid := 1, [1589].log_data[3].valid := 1, [1589].log_data[4].valid := 1, [1589].time.Year := 2022, [1589].time.Month := 4, [1589].time.Day := 29, [1589].time.Hour := 9, [1589].time.Minute := 59, [1589].time.Second := 59, [1589].time.DST_ON := 1, [1590].log_data[0].min := 1.0, [1590].log_data[0].max := 1.0, [1590].log_data[0].total := 300.0, [1590].log_data[0].time := 300.0, [1590].log_data[0].valid := 1, [1590].log_data[1].valid := 1, [1590].log_data[2].valid := 1, [1590].log_data[3].valid := 1, [1590].log_data[4].valid := 1, [1590].time.Year := 2022, [1590].time.Month := 4, [1590].time.Day := 29, [1590].time.Hour := 10, [1590].time.Minute := 4, [1590].time.Second := 59, [1590].time.DST_ON := 1, [1591].log_data[0].min := 1.0, [1591].log_data[0].max := 1.0, [1591].log_data[0].total := 300.001, [1591].log_data[0].time := 300.001, [1591].log_data[0].minminute := 5, [1591].log_data[0].maxminute := 5, [1591].log_data[0].valid := 1, [1591].log_data[1].valid := 1, [1591].log_data[2].valid := 1, [1591].log_data[3].valid := 1, [1591].log_data[4].valid := 1, [1591].time.Year := 2022, [1591].time.Month := 4, [1591].time.Day := 29, [1591].time.Hour := 10,
        [1591].time.Minute := 9, [1591].time.Second := 59, [1591].time.DST_ON := 1, [1592].log_data[0].min := 1.0, [1592].log_data[0].max := 1.0, [1592].log_data[0].total := 300.0, [1592].log_data[0].time := 300.0, [1592].log_data[0].minminute := 10, [1592].log_data[0].maxminute := 10, [1592].log_data[0].valid := 1, [1592].log_data[1].valid := 1, [1592].log_data[2].valid := 1, [1592].log_data[3].valid := 1, [1592].log_data[4].valid := 1, [1592].time.Year := 2022, [1592].time.Month := 4, [1592].time.Day := 29, [1592].time.Hour := 10, [1592].time.Minute := 14, [1592].time.Second := 59, [1592].time.DST_ON := 1, [1593].log_data[0].min := 1.0, [1593].log_data[0].max := 1.0, [1593].log_data[0].total := 300.0, [1593].log_data[0].time := 300.0, [1593].log_data[0].minminute := 15, [1593].log_data[0].maxminute := 15, [1593].log_data[0].valid := 1, [1593].log_data[1].valid := 1, [1593].log_data[2].valid := 1, [1593].log_data[3].valid := 1, [1593].log_data[4].valid := 1, [1593].time.Year := 2022, [1593].time.Month := 4, [1593].time.Day := 29, [1593].time.Hour := 10, [1593].time.Minute := 19, [1593].time.Second := 59, [1593].time.DST_ON := 1, [1594].log_data[0].min := 1.0, [1594].log_data[0].max := 1.0, [1594].log_data[0].total := 300.0, [1594].log_data[0].time := 300.0, [1594].log_data[0].minminute := 20, [1594].log_data[0].maxminute := 20, [1594].log_data[0].valid := 1, [1594].log_data[1].valid := 1, [1594].log_data[2].valid := 1, [1594].log_data[3].valid := 1, [1594].log_data[4].valid := 1, [1594].time.Year := 2022, [1594].time.Month := 4, [1594].time.Day := 29, [1594].time.Hour := 10, [1594].time.Minute := 24, [1594].time.Second := 59, [1594].time.DST_ON := 1, [1595].log_data[0].min := 1.0, [1595].log_data[0].max := 1.0, [1595].log_data[0].total := 300.0,
        [1595].log_data[0].time := 300.0, [1595].log_data[0].minminute := 25, [1595].log_data[0].maxminute := 25, [1595].log_data[0].valid := 1, [1595].log_data[1].valid := 1, [1595].log_data[2].valid := 1, [1595].log_data[3].valid := 1, [1595].log_data[4].valid := 1, [1595].time.Year := 2022, [1595].time.Month := 4, [1595].time.Day := 29, [1595].time.Hour := 10, [1595].time.Minute := 29, [1595].time.Second := 59, [1595].time.DST_ON := 1, [1596].log_data[0].min := 1.0, [1596].log_data[0].max := 1.0, [1596].log_data[0].total := 300.0, [1596].log_data[0].time := 300.0, [1596].log_data[0].minminute := 30, [1596].log_data[0].maxminute := 30, [1596].log_data[0].valid := 1, [1596].log_data[1].valid := 1, [1596].log_data[2].valid := 1, [1596].log_data[3].valid := 1, [1596].log_data[4].valid := 1, [1596].time.Year := 2022, [1596].time.Month := 4, [1596].time.Day := 29, [1596].time.Hour := 10, [1596].time.Minute := 34, [1596].time.Second := 59, [1596].time.DST_ON := 1, [1597].log_data[0].min := 1.0, [1597].log_data[0].max := 1.0, [1597].log_data[0].total := 300.0, [1597].log_data[0].time := 300.0, [1597].log_data[0].minminute := 35, [1597].log_data[0].maxminute := 35, [1597].log_data[0].valid := 1, [1597].log_data[1].valid := 1, [1597].log_data[2].valid := 1, [1597].log_data[3].valid := 1, [1597].log_data[4].valid := 1, [1597].time.Year := 2022, [1597].time.Month := 4, [1597].time.Day := 29, [1597].time.Hour := 10, [1597].time.Minute := 39, [1597].time.Second := 59, [1597].time.DST_ON := 1, [1598].log_data[0].min := 1.0, [1598].log_data[0].max := 1.0, [1598].log_data[0].total := 300.0, [1598].log_data[0].time := 300.0, [1598].log_data[0].minminute := 40, [1598].log_data[0].maxminute := 40, [1598].log_data[0].valid := 1, [1598].log_data[1].valid := 1, [1598].log_data[2].valid := 1,
        [1598].log_data[3].valid := 1, [1598].log_data[4].valid := 1, [1598].time.Year := 2022, [1598].time.Month := 4, [1598].time.Day := 29, [1598].time.Hour := 10, [1598].time.Minute := 44, [1598].time.Second := 59, [1598].time.DST_ON := 1, [1599].log_data[0].min := 1.0, [1599].log_data[0].max := 1.0, [1599].log_data[0].total := 300.0, [1599].log_data[0].time := 300.0, [1599].log_data[0].minminute := 45, [1599].log_data[0].maxminute := 45, [1599].log_data[0].valid := 1, [1599].log_data[1].valid := 1, [1599].log_data[2].valid := 1, [1599].log_data[3].valid := 1, [1599].log_data[4].valid := 1, [1599].time.Year := 2022, [1599].time.Month := 4, [1599].time.Day := 29, [1599].time.Hour := 10, [1599].time.Minute := 49, [1599].time.Second := 59, [1599].time.DST_ON := 1, [1600].log_data[0].min := 1.0, [1600].log_data[0].max := 1.0, [1600].log_data[0].total := 300.0, [1600].log_data[0].time := 300.0, [1600].log_data[0].minminute := 50, [1600].log_data[0].maxminute := 50, [1600].log_data[0].valid := 1, [1600].log_data[1].valid := 1, [1600].log_data[2].valid := 1, [1600].log_data[3].valid := 1, [1600].log_data[4].valid := 1, [1600].time.Year := 2022, [1600].time.Month := 4, [1600].time.Day := 29, [1600].time.Hour := 10, [1600].time.Minute := 54, [1600].time.Second := 59, [1600].time.DST_ON := 1, [1601].log_data[0].min := 1.0, [1601].log_data[0].max := 1.0, [1601].log_data[0].total := 300.0, [1601].log_data[0].time := 300.0, [1601].log_data[0].minminute := 55, [1601].log_data[0].maxminute := 55, [1601].log_data[0].valid := 1, [1601].log_data[1].valid := 1, [1601].log_data[2].valid := 1, [1601].log_data[3].valid := 1, [1601].log_data[4].valid := 1, [1601].time.Year := 2022, [1601].time.Month := 4, [1601].time.Day := 29, [1601].time.Hour := 10,
        [1601].time.Minute := 59, [1601].time.Second := 59, [1601].time.DST_ON := 1, [1602].log_data[0].min := 1.0, [1602].log_data[0].max := 1.0, [1602].log_data[0].total := 300.0, [1602].log_data[0].time := 300.0, [1602].log_data[0].valid := 1, [1602].log_data[1].valid := 1, [1602].log_data[2].valid := 1, [1602].log_data[3].valid := 1, [1602].log_data[4].valid := 1, [1602].time.Year := 2022, [1602].time.Month := 4, [1602].time.Day := 29, [1602].time.Hour := 11, [1602].time.Minute := 4, [1602].time.Second := 59, [1602].time.DST_ON := 1, [1603].log_data[0].min := 1.0, [1603].log_data[0].max := 1.0, [1603].log_data[0].total := 300.0, [1603].log_data[0].time := 300.0, [1603].log_data[0].minminute := 5, [1603].log_data[0].maxminute := 5, [1603].log_data[0].valid := 1, [1603].log_data[1].valid := 1, [1603].log_data[2].valid := 1, [1603].log_data[3].valid := 1, [1603].log_data[4].valid := 1, [1603].time.Year := 2022, [1603].time.Month := 4, [1603].time.Day := 29, [1603].time.Hour := 11, [1603].time.Minute := 9, [1603].time.Second := 59, [1603].time.DST_ON := 1, [1604].log_data[0].min := 1.0, [1604].log_data[0].max := 1.0, [1604].log_data[0].total := 300.0, [1604].log_data[0].time := 300.0, [1604].log_data[0].minminute := 10, [1604].log_data[0].maxminute := 10, [1604].log_data[0].valid := 1, [1604].log_data[1].valid := 1, [1604].log_data[2].valid := 1, [1604].log_data[3].valid := 1, [1604].log_data[4].valid := 1, [1604].time.Year := 2022, [1604].time.Month := 4, [1604].time.Day := 29, [1604].time.Hour := 11, [1604].time.Minute := 14, [1604].time.Second := 59, [1604].time.DST_ON := 1, [1605].log_data[0].min := 1.0, [1605].log_data[0].max := 1.0, [1605].log_data[0].total := 300.0, [1605].log_data[0].time := 300.0, [1605].log_data[0].minminute := 15,
        [1605].log_data[0].maxminute := 15, [1605].log_data[0].valid := 1, [1605].log_data[1].valid := 1, [1605].log_data[2].valid := 1, [1605].log_data[3].valid := 1, [1605].log_data[4].valid := 1, [1605].time.Year := 2022, [1605].time.Month := 4, [1605].time.Day := 29, [1605].time.Hour := 11, [1605].time.Minute := 19, [1605].time.Second := 59, [1605].time.DST_ON := 1, [1606].log_data[0].min := 1.0, [1606].log_data[0].max := 1.0, [1606].log_data[0].total := 300.0, [1606].log_data[0].time := 300.0, [1606].log_data[0].minminute := 20, [1606].log_data[0].maxminute := 20, [1606].log_data[0].valid := 1, [1606].log_data[1].valid := 1, [1606].log_data[2].valid := 1, [1606].log_data[3].valid := 1, [1606].log_data[4].valid := 1, [1606].time.Year := 2022, [1606].time.Month := 4, [1606].time.Day := 29, [1606].time.Hour := 11, [1606].time.Minute := 24, [1606].time.Second := 59, [1606].time.DST_ON := 1, [1607].log_data[0].min := 1.0, [1607].log_data[0].max := 1.0, [1607].log_data[0].total := 300.0, [1607].log_data[0].time := 300.0, [1607].log_data[0].minminute := 25, [1607].log_data[0].maxminute := 25, [1607].log_data[0].valid := 1, [1607].log_data[1].valid := 1, [1607].log_data[2].valid := 1, [1607].log_data[3].valid := 1, [1607].log_data[4].valid := 1, [1607].time.Year := 2022, [1607].time.Month := 4, [1607].time.Day := 29, [1607].time.Hour := 11, [1607].time.Minute := 29, [1607].time.Second := 59, [1607].time.DST_ON := 1, [1608].log_data[0].min := 1.0, [1608].log_data[0].max := 1.0, [1608].log_data[0].total := 300.0, [1608].log_data[0].time := 300.0, [1608].log_data[0].minminute := 30, [1608].log_data[0].maxminute := 30, [1608].log_data[0].valid := 1, [1608].log_data[1].valid := 1, [1608].log_data[2].valid := 1, [1608].log_data[3].valid := 1, [1608].log_data[4].valid := 1,
        [1608].time.Year := 2022, [1608].time.Month := 4, [1608].time.Day := 29, [1608].time.Hour := 11, [1608].time.Minute := 34, [1608].time.Second := 59, [1608].time.DST_ON := 1, [1609].log_data[0].min := 1.0, [1609].log_data[0].max := 1.0, [1609].log_data[0].total := 300.0, [1609].log_data[0].time := 300.0, [1609].log_data[0].minminute := 35, [1609].log_data[0].maxminute := 35, [1609].log_data[0].valid := 1, [1609].log_data[1].valid := 1, [1609].log_data[2].valid := 1, [1609].log_data[3].valid := 1, [1609].log_data[4].valid := 1, [1609].time.Year := 2022, [1609].time.Month := 4, [1609].time.Day := 29, [1609].time.Hour := 11, [1609].time.Minute := 39, [1609].time.Second := 59, [1609].time.DST_ON := 1, [1610].log_data[0].min := 1.0, [1610].log_data[0].max := 1.0, [1610].log_data[0].total := 300.0, [1610].log_data[0].time := 300.0, [1610].log_data[0].minminute := 40, [1610].log_data[0].maxminute := 40, [1610].log_data[0].valid := 1, [1610].log_data[1].valid := 1, [1610].log_data[2].valid := 1, [1610].log_data[3].valid := 1, [1610].log_data[4].valid := 1, [1610].time.Year := 2022, [1610].time.Month := 4, [1610].time.Day := 29, [1610].time.Hour := 11, [1610].time.Minute := 44, [1610].time.Second := 59, [1610].time.DST_ON := 1, [1611].log_data[0].min := 1.0, [1611].log_data[0].max := 1.0, [1611].log_data[0].total := 300.0, [1611].log_data[0].time := 300.0, [1611].log_data[0].minminute := 45, [1611].log_data[0].maxminute := 45, [1611].log_data[0].valid := 1, [1611].log_data[1].valid := 1, [1611].log_data[2].valid := 1, [1611].log_data[3].valid := 1, [1611].log_data[4].valid := 1, [1611].time.Year := 2022, [1611].time.Month := 4, [1611].time.Day := 29, [1611].time.Hour := 11, [1611].time.Minute := 49, [1611].time.Second := 59,
        [1611].time.DST_ON := 1, [1612].log_data[0].min := 1.0, [1612].log_data[0].max := 1.0, [1612].log_data[0].total := 300.0, [1612].log_data[0].time := 300.0, [1612].log_data[0].minminute := 50, [1612].log_data[0].maxminute := 50, [1612].log_data[0].valid := 1, [1612].log_data[1].valid := 1, [1612].log_data[2].valid := 1, [1612].log_data[3].valid := 1, [1612].log_data[4].valid := 1, [1612].time.Year := 2022, [1612].time.Month := 4, [1612].time.Day := 29, [1612].time.Hour := 11, [1612].time.Minute := 54, [1612].time.Second := 59, [1612].time.DST_ON := 1, [1613].log_data[0].min := 1.0, [1613].log_data[0].max := 1.0, [1613].log_data[0].total := 300.0, [1613].log_data[0].time := 300.0, [1613].log_data[0].minminute := 55, [1613].log_data[0].maxminute := 55, [1613].log_data[0].valid := 1, [1613].log_data[1].valid := 1, [1613].log_data[2].valid := 1, [1613].log_data[3].valid := 1, [1613].log_data[4].valid := 1, [1613].time.Year := 2022, [1613].time.Month := 4, [1613].time.Day := 29, [1613].time.Hour := 11, [1613].time.Minute := 59, [1613].time.Second := 59, [1613].time.DST_ON := 1, [1614].log_data[0].min := 1.0, [1614].log_data[0].max := 1.0, [1614].log_data[0].total := 300.0, [1614].log_data[0].time := 300.0, [1614].log_data[0].valid := 1, [1614].log_data[1].valid := 1, [1614].log_data[2].valid := 1, [1614].log_data[3].valid := 1, [1614].log_data[4].valid := 1, [1614].time.Year := 2022, [1614].time.Month := 4, [1614].time.Day := 29, [1614].time.Hour := 12, [1614].time.Minute := 4, [1614].time.Second := 59, [1614].time.DST_ON := 1, [1615].log_data[0].min := 1.0, [1615].log_data[0].max := 1.0, [1615].log_data[0].total := 300.0, [1615].log_data[0].time := 300.0, [1615].log_data[0].minminute := 5, [1615].log_data[0].maxminute := 5, [1615].log_data[0].valid := 1,
        [1615].log_data[1].valid := 1, [1615].log_data[2].valid := 1, [1615].log_data[3].valid := 1, [1615].log_data[4].valid := 1, [1615].time.Year := 2022, [1615].time.Month := 4, [1615].time.Day := 29, [1615].time.Hour := 12, [1615].time.Minute := 9, [1615].time.Second := 59, [1615].time.DST_ON := 1, [1616].log_data[0].min := 1.0, [1616].log_data[0].max := 1.0, [1616].log_data[0].total := 300.0, [1616].log_data[0].time := 300.0, [1616].log_data[0].minminute := 10, [1616].log_data[0].maxminute := 10, [1616].log_data[0].valid := 1, [1616].log_data[1].valid := 1, [1616].log_data[2].valid := 1, [1616].log_data[3].valid := 1, [1616].log_data[4].valid := 1, [1616].time.Year := 2022, [1616].time.Month := 4, [1616].time.Day := 29, [1616].time.Hour := 12, [1616].time.Minute := 14, [1616].time.Second := 59, [1616].time.DST_ON := 1, [1617].log_data[0].min := 1.0, [1617].log_data[0].max := 1.0, [1617].log_data[0].total := 300.0, [1617].log_data[0].time := 300.0, [1617].log_data[0].minminute := 15, [1617].log_data[0].maxminute := 15, [1617].log_data[0].valid := 1, [1617].log_data[1].valid := 1, [1617].log_data[2].valid := 1, [1617].log_data[3].valid := 1, [1617].log_data[4].valid := 1, [1617].time.Year := 2022, [1617].time.Month := 4, [1617].time.Day := 29, [1617].time.Hour := 12, [1617].time.Minute := 19, [1617].time.Second := 59, [1617].time.DST_ON := 1, [1618].log_data[0].min := 1.0, [1618].log_data[0].max := 1.0, [1618].log_data[0].total := 300.0, [1618].log_data[0].time := 300.0, [1618].log_data[0].minminute := 20, [1618].log_data[0].maxminute := 20, [1618].log_data[0].valid := 1, [1618].log_data[1].valid := 1, [1618].log_data[2].valid := 1, [1618].log_data[3].valid := 1, [1618].log_data[4].valid := 1, [1618].time.Year := 2022, [1618].time.Month := 4,
